C05459=1058.645,309.045,397.535,173.307,35.654,156.681
C05460=1058.639,308.797,397.568,173.303,35.650,156.680
C05461=1058.631,308.551,397.601,173.300,35.645,156.679
C05462=1058.625,308.302,397.633,173.297,35.642,156.679
C05463=1058.618,308.054,397.666,173.293,35.638,156.678
C05464=1058.612,307.806,397.699,173.290,35.634,156.677
C05465=1058.606,307.559,397.731,173.287,35.630,156.676
C05466=1058.600,307.311,397.764,173.283,35.626,156.675
C05467=1058.593,307.064,397.797,173.280,35.622,156.674
C05468=1058.586,306.815,397.830,173.277,35.617,156.673
C05469=1058.579,306.568,397.862,173.274,35.613,156.672
C05470=1058.573,306.320,397.895,173.271,35.609,156.672
C05471=1058.567,306.073,397.928,173.267,35.605,156.671
C05472=1058.560,305.825,397.960,173.264,35.601,156.670
C05473=1058.554,305.578,397.993,173.260,35.598,156.669
C05474=1058.548,305.329,398.025,173.257,35.594,156.668
C05475=1058.541,305.081,398.058,173.255,35.590,156.667
C05476=1058.534,304.834,398.090,173.251,35.585,156.666
C05477=1058.528,304.586,398.123,173.248,35.581,156.666
C05478=1058.522,304.338,398.155,173.244,35.577,156.665
C05479=1058.515,304.090,398.188,173.241,35.573,156.664
C05480=1058.509,303.842,398.220,173.238,35.569,156.663
C05481=1058.503,303.593,398.254,173.234,35.566,156.662
C05482=1058.496,303.345,398.285,173.232,35.561,156.661
C05483=1058.490,303.097,398.318,173.228,35.557,156.660
C05484=1058.484,302.850,398.351,173.225,35.553,156.660
C05485=1058.478,302.602,398.383,173.222,35.549,156.659
C05486=1058.471,302.354,398.416,173.218,35.545,156.658
C05487=1058.464,302.107,398.448,173.216,35.541,156.657
C05488=1058.458,301.859,398.480,173.213,35.538,156.656
C05489=1058.452,301.611,398.513,173.209,35.533,156.655
C05490=1058.446,301.363,398.545,173.206,35.529,156.655
C05491=1058.440,301.115,398.577,173.202,35.525,156.654
C05492=1058.433,300.867,398.609,173.200,35.521,156.653
C05493=1058.427,300.620,398.642,173.197,35.517,156.652
C05494=1058.420,300.372,398.674,173.193,35.514,156.651
C05495=1058.414,300.124,398.706,173.190,35.509,156.650
C05496=1058.408,299.876,398.739,173.187,35.505,156.649
C05497=1058.401,299.628,398.770,173.184,35.501,156.649
C05498=1058.395,299.380,398.802,173.181,35.497,156.648
C05499=1058.389,299.133,398.835,173.177,35.494,156.647
C05500=1058.383,298.884,398.867,173.174,35.490,156.646
C05501=1058.377,298.638,398.899,173.172,35.485,156.645
C05502=1058.371,298.390,398.931,173.168,35.481,156.644
C05503=1058.364,298.142,398.964,173.165,35.477,156.644
C05504=1058.358,297.894,398.996,173.162,35.474,156.643
C05505=1058.352,297.646,399.027,173.159,35.470,156.642
C05506=1058.345,297.398,399.060,173.156,35.466,156.641
C05507=1058.339,297.150,399.092,173.152,35.461,156.640
C05508=1058.334,296.903,399.124,173.150,35.457,156.639
C05509=1058.327,296.655,399.156,173.147,35.454,156.639
C05510=1058.321,296.407,399.188,173.143,35.450,156.638
C05511=1058.314,296.159,399.219,173.140,35.446,156.637
C05512=1058.308,295.911,399.251,173.138,35.442,156.636
C05513=1058.302,295.663,399.283,173.134,35.438,156.635
C05514=1058.295,295.415,399.315,173.131,35.434,156.635
C05515=1058.289,295.168,399.347,173.128,35.430,156.634
C05516=1058.283,294.919,399.379,173.125,35.426,156.633
C05517=1058.276,294.672,399.410,173.122,35.423,156.632
C05518=1058.270,294.424,399.441,173.119,35.419,156.631
C05519=1058.264,294.176,399.473,173.115,35.415,156.630
C05520=1058.257,293.928,399.505,173.113,35.411,156.630
C05521=1058.250,293.680,399.536,173.110,35.407,156.629
C05522=1058.244,293.432,399.568,173.106,35.403,156.628
C05523=1058.238,293.185,399.599,173.104,35.399,156.627
C05524=1058.232,292.937,399.631,173.101,35.396,156.626
C05525=1058.226,292.689,399.663,173.097,35.392,156.626
C05526=1058.219,292.441,399.694,173.095,35.388,156.625
C05527=1058.213,292.193,399.726,173.092,35.384,156.624
C05528=1058.206,291.945,399.758,173.088,35.380,156.623
C05529=1058.200,291.697,399.789,173.086,35.376,156.622
C05530=1058.194,291.457,399.820,173.083,35.373,156.622
C05531=1058.188,291.217,399.850,173.079,35.369,156.621
C05532=1058.182,290.976,399.881,173.077,35.365,156.620
C05533=1058.175,290.736,399.911,173.074,35.362,156.619
C05534=1058.169,290.496,399.942,173.071,35.358,156.619
C05535=1058.163,290.255,399.972,173.068,35.354,156.618
C05536=1058.156,290.015,400.002,173.065,35.350,156.617
C05537=1058.151,289.774,400.033,173.062,35.347,156.616
C05538=1058.144,289.527,400.064,173.059,35.343,156.615
C05539=1058.138,289.279,400.095,173.057,35.339,156.615
C05540=1058.132,289.031,400.128,173.053,35.335,156.614
C05541=1058.126,288.783,400.158,173.050,35.332,156.613
C05542=1058.119,288.535,400.189,173.048,35.327,156.612
C05543=1058.112,288.287,400.221,173.044,35.324,156.611
C05544=1058.106,288.039,400.251,173.041,35.320,156.611
C05545=1058.100,287.791,400.283,173.039,35.316,156.610
C05546=1058.094,287.543,400.315,173.035,35.313,156.609
C05547=1058.088,287.295,400.345,173.032,35.309,156.608
C05548=1058.081,287.047,400.377,173.030,35.305,156.607
C05549=1058.075,286.800,400.408,173.026,35.301,156.607
C05550=1058.068,286.551,400.438,173.024,35.297,156.606
C05551=1058.062,286.303,400.470,173.021,35.294,156.605
C05552=1058.056,286.055,400.500,173.017,35.290,156.604
C05553=1058.049,285.807,400.532,173.015,35.286,156.604
C05554=1058.042,285.560,400.563,173.012,35.282,156.603
C05555=1058.036,285.312,400.593,173.008,35.278,156.602
C05556=1058.030,285.064,400.625,173.006,35.275,156.601
C05557=1058.023,284.815,400.656,173.003,35.271,156.600
C05558=1058.017,284.568,400.687,173.001,35.267,156.600
C05559=1058.011,284.320,400.717,172.997,35.263,156.599
C05560=1058.004,284.071,400.748,172.994,35.260,156.598
C05561=1057.998,283.824,400.779,172.992,35.256,156.597
C05562=1057.992,283.575,400.810,172.988,35.252,156.596
C05563=1057.986,283.328,400.841,172.986,35.248,156.596
C05564=1057.979,283.080,400.872,172.983,35.245,156.595
C05565=1057.973,282.832,400.903,172.980,35.241,156.594
C05566=1057.967,282.584,400.933,172.977,35.237,156.593
C05567=1057.960,282.335,400.964,172.974,35.233,156.593
C05568=1057.954,282.088,400.995,172.971,35.229,156.592
C05569=1057.948,281.840,401.026,172.968,35.226,156.591
C05570=1057.942,281.592,401.056,172.966,35.222,156.590
C05571=1057.935,281.344,401.088,172.962,35.218,156.590
C05572=1057.929,281.096,401.118,172.960,35.215,156.589
C05573=1057.923,280.848,401.149,172.957,35.210,156.588
C05574=1057.917,280.600,401.179,172.955,35.207,156.587
C05575=1057.910,280.352,401.211,172.951,35.203,156.586
C05576=1057.905,280.104,401.241,172.949,35.199,156.586
C05577=1057.898,279.856,401.272,172.946,35.196,156.585
C05578=1057.892,279.608,401.302,172.942,35.192,156.584
C05579=1057.885,279.359,401.332,172.940,35.188,156.583
C05580=1057.879,279.112,401.364,172.937,35.184,156.583
C05581=1057.873,278.864,401.394,172.934,35.181,156.582
C05582=1057.866,278.615,401.425,172.931,35.177,156.581
C05583=1057.860,278.368,401.454,172.929,35.173,156.580
C05584=1057.853,278.119,401.485,172.926,35.170,156.580
C05585=1057.847,277.871,401.515,172.923,35.165,156.579
C05586=1057.842,277.637,401.544,172.920,35.162,156.578
C05587=1057.836,277.401,401.573,172.918,35.159,156.577
C05588=1057.830,277.166,401.602,172.915,35.155,156.577
C05589=1057.824,276.932,401.631,172.912,35.152,156.576
C05590=1057.817,276.697,401.659,172.910,35.148,156.575
C05591=1057.811,276.462,401.688,172.907,35.145,156.574
C05592=1057.806,276.227,401.717,172.904,35.141,156.574
C05593=1057.800,275.992,401.745,172.902,35.138,156.573
C05594=1057.794,275.744,401.776,172.899,35.134,156.572
C05595=1057.787,275.496,401.806,172.896,35.130,156.571
C05596=1057.781,275.248,401.837,172.893,35.126,156.571
C05597=1057.775,275.000,401.867,172.891,35.123,156.570
C05598=1057.764,274.601,401.916,172.886,35.117,156.569
C05599=1057.754,274.203,401.964,172.882,35.111,156.568
C05600=1057.744,273.805,402.012,172.877,35.105,156.566
C05601=1057.734,273.406,402.060,172.873,35.099,156.565
C05602=1057.728,273.158,402.091,172.870,35.095,156.564
C05603=1057.722,272.911,402.121,172.867,35.091,156.564
C05604=1057.715,272.662,402.151,172.865,35.088,156.563
C05605=1057.710,272.414,402.181,172.862,35.084,156.562
C05606=1057.703,272.166,402.211,172.860,35.081,156.561
C05607=1057.697,271.918,402.241,172.856,35.076,156.560
C05608=1057.690,271.670,402.270,172.854,35.073,156.560
C05609=1057.684,271.421,402.301,172.851,35.069,156.559
C05610=1057.678,271.173,402.331,172.849,35.066,156.558
C05611=1057.672,270.926,402.361,172.845,35.062,156.558
C05612=1057.665,270.677,402.391,172.843,35.058,156.557
C05613=1057.659,270.429,402.421,172.841,35.054,156.556
C05614=1057.653,270.181,402.450,172.837,35.051,156.555
C05615=1057.646,269.933,402.481,172.835,35.047,156.555
C05616=1057.640,269.685,402.510,172.832,35.044,156.554
C05617=1057.634,269.437,402.540,172.830,35.040,156.553
C05618=1057.627,269.188,402.570,172.826,35.036,156.552
C05619=1057.621,268.940,402.600,172.824,35.032,156.552
C05620=1057.615,268.692,402.630,172.822,35.029,156.551
C05621=1057.609,268.444,402.659,172.818,35.025,156.550
C05622=1057.602,268.196,402.689,172.816,35.021,156.549
C05623=1057.596,267.948,402.718,172.813,35.018,156.549
C05624=1057.590,267.700,402.749,172.811,35.014,156.548
C05625=1057.583,267.451,402.778,172.808,35.010,156.547
C05626=1057.577,267.204,402.808,172.805,35.007,156.546
C05627=1057.571,266.955,402.838,172.803,35.003,156.546
C05628=1057.565,266.708,402.867,172.800,35.000,156.545
C05629=1057.558,266.459,402.897,172.797,34.995,156.544
C05630=1057.552,266.210,402.926,172.795,34.992,156.543
C05631=1057.546,265.963,402.956,172.792,34.988,156.543
C05632=1057.540,265.715,402.985,172.790,34.985,156.542
C05633=1057.533,265.466,403.016,172.786,34.981,156.541
C05634=1057.527,265.218,403.045,172.784,34.978,156.540
C05635=1057.521,264.970,403.074,172.782,34.973,156.540
C05636=1057.515,264.722,403.104,172.778,34.970,156.539
C05637=1057.509,264.474,403.133,172.776,34.966,156.538
C05638=1057.502,264.225,403.163,172.774,34.963,156.537
C05639=1057.496,263.977,403.192,172.771,34.959,156.537
C05640=1057.490,263.729,403.222,172.768,34.956,156.536
C05641=1057.483,263.481,403.251,172.766,34.951,156.535
C05642=1057.476,263.165,403.288,172.763,34.947,156.534
C05643=1057.468,262.850,403.326,172.760,34.942,156.533
C05644=1057.460,262.534,403.363,172.756,34.938,156.532
C05645=1057.451,262.219,403.400,172.753,34.933,156.532
C05646=1057.444,261.971,403.430,172.750,34.930,156.531
C05647=1057.438,261.722,403.459,172.747,34.926,156.530
C05648=1057.432,261.474,403.488,172.745,34.923,156.529
C05649=1057.425,261.226,403.517,172.742,34.919,156.529
C05650=1057.418,260.977,403.546,172.740,34.915,156.528
C05651=1057.412,260.729,403.575,172.737,34.912,156.527
C05652=1057.406,260.481,403.604,172.734,34.908,156.526
C05653=1057.400,260.233,403.633,172.732,34.905,156.526
C05654=1057.393,259.985,403.662,172.730,34.901,156.525
C05655=1057.387,259.737,403.691,172.726,34.897,156.524
C05656=1057.380,259.488,403.721,172.724,34.893,156.523
C05657=1057.374,259.240,403.750,172.722,34.890,156.523
C05658=1057.368,258.992,403.779,172.719,34.886,156.522
C05659=1057.362,258.743,403.808,172.716,34.883,156.521
C05660=1057.355,258.495,403.837,172.714,34.879,156.521
C05661=1057.349,258.247,403.866,172.711,34.875,156.520
C05662=1057.343,257.999,403.895,172.709,34.872,156.519
C05663=1057.336,257.751,403.923,172.706,34.868,156.518
C05664=1057.329,257.502,403.953,172.703,34.865,156.518
C05665=1057.323,257.254,403.981,172.701,34.861,156.517
C05666=1057.317,257.006,404.010,172.699,34.857,156.516
C05667=1057.311,256.757,404.039,172.695,34.854,156.516
C05668=1057.304,256.509,404.068,172.693,34.850,156.515
C05669=1057.298,256.261,404.097,172.691,34.847,156.514
C05670=1057.292,256.013,404.126,172.689,34.843,156.513
C05671=1057.286,255.765,404.155,172.685,34.839,156.513
C05672=1057.280,255.516,404.184,172.683,34.836,156.512
C05673=1057.273,255.268,404.213,172.681,34.832,156.511
C05674=1057.266,255.020,404.241,172.679,34.828,156.510
C05675=1057.260,254.772,404.270,172.675,34.825,156.510
C05676=1057.254,254.523,404.299,172.673,34.821,156.509
C05677=1057.248,254.275,404.328,172.671,34.817,156.508
C05678=1057.242,254.027,404.357,172.669,34.814,156.508
C05679=1057.235,253.779,404.386,172.666,34.810,156.507
C05680=1057.230,253.530,404.414,172.663,34.807,156.506
C05681=1057.223,253.282,404.443,172.661,34.803,156.505
C05682=1057.217,253.034,404.472,172.659,34.799,156.505
C05683=1057.210,252.785,404.500,172.656,34.796,156.504
C05684=1057.204,252.537,404.529,172.653,34.792,156.503
C05685=1057.198,252.289,404.557,172.651,34.788,156.502
C05686=1057.192,252.040,404.586,172.649,34.784,156.502
C05687=1057.186,251.792,404.615,172.646,34.781,156.501
C05688=1057.180,251.544,404.644,172.643,34.777,156.500
C05689=1057.173,251.295,404.673,172.641,34.774,156.500
C05690=1057.167,251.047,404.700,172.639,34.770,156.499
C05691=1057.161,250.799,404.729,172.637,34.766,156.498
C05692=1057.155,250.551,404.758,172.633,34.762,156.497
C05693=1057.149,250.303,404.786,172.631,34.759,156.497
C05694=1057.143,250.068,404.814,172.629,34.755,156.496
C05695=1057.137,249.835,404.841,172.627,34.752,156.495
C05696=1057.131,249.601,404.868,172.625,34.748,156.494
C05697=1057.125,249.367,404.894,172.622,34.745,156.494
C05698=1057.120,249.133,404.921,172.620,34.741,156.493
C05699=1057.114,248.900,404.948,172.618,34.738,156.492
C05700=1057.108,248.665,404.975,172.616,34.735,156.492
C05701=1057.103,248.431,405.002,172.613,34.731,156.491
C05702=1057.096,248.183,405.030,172.611,34.727,156.490
C05703=1057.090,247.935,405.058,172.608,34.724,156.490
C05704=1057.084,247.686,405.087,172.606,34.720,156.489
C05705=1057.078,247.438,405.116,172.604,34.716,156.488
C05706=1057.072,247.189,405.144,172.601,34.712,156.487
C05707=1057.066,246.941,405.172,172.599,34.709,156.487
C05708=1057.060,246.694,405.201,172.597,34.705,156.486
C05709=1057.054,246.445,405.229,172.594,34.701,156.485
C05710=1057.048,246.196,405.257,172.591,34.697,156.484
C05711=1057.041,245.948,405.286,172.589,34.694,156.484
C05712=1057.035,245.699,405.314,172.587,34.690,156.483
C05713=1057.029,245.451,405.342,172.585,34.687,156.482
C05714=1057.023,245.203,405.370,172.583,34.683,156.481
C05715=1057.017,244.955,405.399,172.579,34.679,156.481
C05716=1057.010,244.706,405.426,172.577,34.676,156.480
C05717=1057.004,244.458,405.455,172.575,34.672,156.479
C05718=1056.998,244.209,405.483,172.573,34.668,156.479
C05719=1056.992,243.961,405.510,172.570,34.664,156.478
C05720=1056.986,243.713,405.539,172.568,34.661,156.477
C05721=1056.979,243.465,405.567,172.566,34.657,156.476
C05722=1056.973,243.216,405.596,172.563,34.654,156.476
C05723=1056.967,242.967,405.623,172.561,34.650,156.475
C05724=1056.961,242.719,405.651,172.558,34.646,156.474
C05725=1056.955,242.471,405.679,172.556,34.643,156.474
C05726=1056.949,242.222,405.707,172.554,34.639,156.473
C05727=1056.942,241.974,405.736,172.552,34.635,156.472
C05728=1056.936,241.726,405.764,172.549,34.631,156.471
C05729=1056.930,241.478,405.791,172.547,34.628,156.471
C05730=1056.924,241.229,405.820,172.544,34.624,156.470
C05731=1056.917,240.981,405.847,172.542,34.620,156.469
C05732=1056.911,240.733,405.875,172.540,34.617,156.468
C05733=1056.905,240.484,405.903,172.537,34.613,156.468
C05734=1056.898,240.236,405.931,172.535,34.610,156.467
C05735=1056.892,239.987,405.959,172.533,34.606,156.466
C05736=1056.886,239.739,405.987,172.531,34.602,156.466
C05737=1056.880,239.490,406.014,172.529,34.599,156.465
C05738=1056.873,239.242,406.041,172.526,34.595,156.464
C05739=1056.867,238.993,406.070,172.523,34.592,156.463
C05740=1056.861,238.745,406.097,172.521,34.588,156.463
C05741=1056.854,238.497,406.125,172.519,34.584,156.462
C05742=1056.849,238.248,406.153,172.516,34.580,156.461
C05743=1056.842,238.000,406.181,172.514,34.577,156.460
C05744=1056.836,237.752,406.208,172.512,34.573,156.460
C05745=1056.829,237.503,406.236,172.510,34.569,156.459
C05746=1056.823,237.254,406.264,172.508,34.566,156.458
C05747=1056.817,237.006,406.291,172.505,34.562,156.458
C05748=1056.811,236.758,406.319,172.503,34.558,156.457
C05749=1056.804,236.509,406.346,172.501,34.555,156.456
C05750=1056.799,236.273,406.372,172.499,34.551,156.455
C05751=1056.792,236.036,406.399,172.497,34.548,156.455
C05752=1056.787,235.799,406.426,172.494,34.544,156.454
C05753=1056.781,235.562,406.452,172.492,34.541,156.453
C05754=1056.775,235.325,406.478,172.490,34.537,156.453
C05755=1056.769,235.088,406.505,172.488,34.534,156.452
C05756=1056.763,234.850,406.530,172.486,34.530,156.451
C05757=1056.758,234.614,406.556,172.484,34.527,156.451
C05758=1056.751,234.365,406.584,172.481,34.523,156.450
C05759=1056.744,234.117,406.612,172.479,34.519,156.449
C05760=1056.739,233.868,406.639,172.477,34.516,156.448
C05761=1056.732,233.620,406.667,172.475,34.512,156.448
C05762=1056.726,233.372,406.694,172.473,34.508,156.447
C05763=1056.720,233.123,406.721,172.470,34.504,156.446
C05764=1056.714,232.875,406.748,172.468,34.501,156.446
C05765=1056.708,232.627,406.777,172.466,34.497,156.445
C05766=1056.702,232.377,406.804,172.464,34.493,156.444
C05767=1056.696,232.130,406.831,172.462,34.490,156.443
C05768=1056.689,231.881,406.858,172.459,34.486,156.443
C05769=1056.683,231.633,406.885,172.457,34.483,156.442
C05770=1056.677,231.384,406.912,172.455,34.479,156.441
C05771=1056.670,231.135,406.940,172.453,34.475,156.440
C05772=1056.664,230.887,406.967,172.451,34.471,156.440
C05773=1056.658,230.639,406.995,172.448,34.467,156.439
C05774=1056.652,230.390,407.021,172.446,34.464,156.438
C05775=1056.645,230.142,407.049,172.444,34.460,156.438
C05776=1056.639,229.893,407.076,172.442,34.457,156.437
C05777=1056.633,229.645,407.104,172.440,34.453,156.436
C05778=1056.628,229.396,407.131,172.437,34.449,156.435
C05779=1056.621,229.148,407.158,172.435,34.445,156.435
C05780=1056.614,228.900,407.184,172.433,34.441,156.434
C05781=1056.608,228.651,407.212,172.431,34.438,156.433
C05782=1056.601,228.402,407.239,172.429,34.434,156.433
C05783=1056.596,228.154,407.266,172.426,34.431,156.432
C05784=1056.589,227.906,407.294,172.424,34.427,156.431
C05785=1056.583,227.657,407.320,172.422,34.423,156.430
C05786=1056.577,227.408,407.347,172.420,34.420,156.430
C05787=1056.570,227.161,407.374,172.418,34.416,156.429
C05788=1056.564,226.912,407.401,172.415,34.412,156.428
C05789=1056.558,226.663,407.428,172.413,34.408,156.427
C05790=1056.551,226.415,407.455,172.411,34.405,156.427
C05791=1056.545,226.167,407.482,172.409,34.401,156.426
C05792=1056.539,225.917,407.509,172.407,34.397,156.425
C05793=1056.533,225.669,407.536,172.405,34.394,156.425
C05794=1056.526,225.421,407.563,172.402,34.390,156.424
C05795=1056.520,225.173,407.589,172.400,34.386,156.423
C05796=1056.514,224.924,407.616,172.398,34.383,156.422
C05797=1056.508,224.675,407.643,172.396,34.379,156.422
C05798=1056.502,224.427,407.670,172.394,34.375,156.421
C05799=1056.495,224.178,407.697,172.391,34.371,156.420
C05800=1056.489,223.930,407.724,172.389,34.368,156.420
C05801=1056.482,223.681,407.751,172.387,34.364,156.419
C05802=1056.477,223.433,407.777,172.385,34.360,156.418
C05803=1056.471,223.185,407.804,172.383,34.356,156.417
C05804=1056.465,222.935,407.831,172.382,34.353,156.417
C05805=1056.459,222.687,407.857,172.379,34.349,156.416
C05806=1056.452,222.446,407.884,172.377,34.345,156.415
C05807=1056.447,222.206,407.910,172.375,34.342,156.414
C05808=1056.440,221.964,407.936,172.373,34.338,156.414
C05809=1056.434,221.724,407.962,172.371,34.335,156.413
C05810=1056.428,221.483,407.988,172.368,34.331,156.412
C05811=1056.423,221.242,408.013,172.366,34.327,156.412
C05812=1056.416,221.001,408.039,172.365,34.324,156.411
C05813=1056.411,220.760,408.065,172.363,34.320,156.410
C05814=1056.404,220.512,408.091,172.361,34.316,156.410
C05815=1056.398,220.263,408.118,172.359,34.313,156.409
C05816=1056.391,220.015,408.144,172.356,34.309,156.408
C05817=1056.385,219.766,408.171,172.354,34.305,156.407
C05818=1056.379,219.518,408.197,172.352,34.301,156.407
C05819=1056.372,219.269,408.224,172.350,34.298,156.406
C05820=1056.366,219.021,408.250,172.348,34.294,156.405
C05821=1056.360,218.773,408.276,172.347,34.290,156.404
C05822=1056.353,218.524,408.304,172.344,34.287,156.404
C05823=1056.347,218.276,408.330,172.342,34.283,156.403
C05824=1056.341,218.027,408.356,172.340,34.279,156.402
C05825=1056.335,217.778,408.383,172.338,34.275,156.402
C05826=1056.329,217.530,408.409,172.336,34.272,156.401
C05827=1056.323,217.281,408.435,172.334,34.268,156.400
C05828=1056.316,217.032,408.462,172.331,34.264,156.399
C05829=1056.310,216.784,408.488,172.329,34.260,156.399
C05830=1056.303,216.536,408.514,172.328,34.257,156.398
C05831=1056.297,216.287,408.541,172.326,34.253,156.397
C05832=1056.291,216.038,408.567,172.324,34.249,156.396
C05833=1056.285,215.790,408.593,172.321,34.246,156.396
C05834=1056.279,215.542,408.619,172.319,34.241,156.395
C05835=1056.272,215.293,408.646,172.317,34.238,156.394
C05836=1056.266,215.044,408.672,172.315,34.234,156.394
C05837=1056.260,214.796,408.698,172.314,34.230,156.393
C05838=1056.254,214.548,408.724,172.312,34.226,156.392
C05839=1056.247,214.299,408.751,172.309,34.223,156.391
C05840=1056.241,214.050,408.777,172.307,34.219,156.391
C05841=1056.235,213.802,408.803,172.305,34.215,156.390
C05842=1056.229,213.554,408.829,172.303,34.211,156.389
C05843=1056.223,213.304,408.856,172.302,34.207,156.388
C05844=1056.217,213.056,408.882,172.300,34.204,156.388
C05845=1056.210,212.808,408.908,172.297,34.200,156.387
C05846=1056.204,212.559,408.934,172.295,34.196,156.386
C05847=1056.198,212.311,408.960,172.293,34.192,156.385
C05848=1056.191,212.062,408.987,172.291,34.189,156.385
C05849=1056.186,211.813,409.013,172.290,34.184,156.384
C05850=1056.179,211.565,409.039,172.288,34.181,156.383
C05851=1056.173,211.316,409.064,172.286,34.177,156.383
C05852=1056.167,211.067,409.091,172.283,34.174,156.382
C05853=1056.160,210.819,409.117,172.281,34.169,156.381
C05854=1056.154,210.570,409.143,172.279,34.166,156.380
C05855=1056.148,210.322,409.169,172.278,34.162,156.380
C05856=1056.142,210.073,409.195,172.276,34.158,156.379
C05857=1056.135,209.824,409.221,172.274,34.154,156.378
C05858=1056.129,209.576,409.247,172.271,34.150,156.377
C05859=1056.123,209.327,409.273,172.269,34.147,156.377
C05860=1056.117,209.079,409.298,172.268,34.143,156.376
C05861=1056.110,208.831,409.324,172.266,34.139,156.375
C05862=1056.104,208.592,409.350,172.264,34.135,156.374
C05863=1056.099,208.354,409.375,172.262,34.132,156.374
C05864=1056.092,208.116,409.399,172.260,34.128,156.373
C05865=1056.087,207.877,409.424,172.258,34.124,156.372
C05866=1056.081,207.639,409.448,172.256,34.121,156.372
C05867=1056.075,207.400,409.473,172.255,34.117,156.371
C05868=1056.069,207.162,409.498,172.253,34.114,156.370
C05869=1056.062,206.924,409.522,172.251,34.110,156.370
C05870=1056.037,205.873,409.627,172.050,34.020,156.356
C05871=1056.031,205.624,409.652,172.048,34.017,156.356
C05872=1056.025,205.376,409.677,172.045,34.014,156.355
C05873=1056.020,205.127,409.702,172.043,34.011,156.355
C05874=1056.013,204.878,409.727,172.041,34.008,156.354
C05875=1056.008,204.630,409.752,172.038,34.005,156.354
C05876=1056.001,204.381,409.776,172.036,34.002,156.353
C05877=1055.996,204.133,409.801,172.034,33.999,156.353
C05878=1055.990,203.884,409.826,172.031,33.996,156.352
C05879=1055.984,203.635,409.851,172.028,33.993,156.352
C05880=1055.978,203.387,409.876,172.026,33.990,156.351
C05881=1055.972,203.138,409.900,172.024,33.987,156.351
C05882=1055.966,202.888,409.925,172.021,33.984,156.350
C05883=1055.961,202.640,409.950,172.019,33.982,156.350
C05884=1055.954,202.391,409.974,172.017,33.978,156.349
C05885=1055.948,202.143,409.999,172.015,33.975,156.348
C05886=1055.943,201.894,410.023,172.012,33.972,156.348
C05887=1055.937,201.645,410.048,172.010,33.970,156.347
C05888=1055.930,201.397,410.072,172.008,33.967,156.347
C05889=1055.924,201.148,410.097,172.005,33.964,156.346
C05890=1055.918,200.899,410.122,172.002,33.961,156.346
C05891=1055.912,200.651,410.146,172.000,33.958,156.345
C05892=1055.906,200.402,410.171,171.998,33.955,156.345
C05893=1055.900,200.153,410.194,171.995,33.953,156.344
C05894=1055.894,199.904,410.219,171.993,33.950,156.344
C05895=1055.888,199.655,410.244,171.991,33.947,156.343
C05896=1055.882,199.407,410.268,171.989,33.944,156.343
C05897=1055.876,199.158,410.293,171.986,33.941,156.342
C05898=1055.870,198.910,410.316,171.984,33.938,156.342
C05899=1055.864,198.661,410.342,171.982,33.936,156.341
C05900=1055.857,198.412,410.366,171.980,33.933,156.341
C05901=1055.852,198.163,410.390,171.976,33.930,156.340
C05902=1055.845,197.914,410.414,171.974,33.927,156.340
C05903=1055.840,197.666,410.438,171.972,33.924,156.339
C05904=1055.834,197.416,410.463,171.970,33.921,156.339
C05905=1055.828,197.169,410.487,171.967,33.919,156.338
C05906=1055.822,196.919,410.512,171.965,33.916,156.338
C05907=1055.815,196.671,410.536,171.963,33.913,156.337
C05908=1055.810,196.422,410.560,171.961,33.910,156.337
C05909=1055.803,196.173,410.584,171.958,33.907,156.336
C05910=1055.798,195.924,410.608,171.956,33.904,156.336
C05911=1055.791,195.675,410.632,171.954,33.902,156.335
C05912=1055.786,195.427,410.657,171.952,33.899,156.335
C05913=1055.779,195.178,410.681,171.949,33.896,156.334
C05914=1055.774,194.929,410.705,171.946,33.893,156.334
C05915=1055.768,194.680,410.729,171.944,33.891,156.333
C05916=1055.762,194.432,410.753,171.942,33.887,156.333
C05917=1055.756,194.183,410.777,171.940,33.885,156.332
C05918=1055.750,193.934,410.801,171.937,33.882,156.332
C05919=1055.744,193.686,410.825,171.935,33.879,156.331
C05920=1055.738,193.437,410.850,171.933,33.876,156.331
C05921=1055.732,193.188,410.873,171.931,33.874,156.330
C05922=1055.726,192.939,410.898,171.929,33.870,156.330
C05923=1055.720,192.691,410.922,171.926,33.868,156.329
C05924=1055.714,192.441,410.946,171.924,33.865,156.329
C05925=1055.708,192.193,410.970,171.922,33.862,156.328
C05926=1055.703,191.945,410.994,171.920,33.860,156.328
C05927=1055.696,191.696,411.018,171.917,33.857,156.327
C05928=1055.691,191.447,411.042,171.915,33.854,156.327
C05929=1055.685,191.198,411.067,171.912,33.851,156.326
C05930=1055.679,190.949,411.091,171.910,33.848,156.326
C05931=1055.673,190.665,411.118,171.908,33.845,156.325
C05932=1055.666,190.381,411.145,171.905,33.842,156.325
C05933=1055.659,190.097,411.173,171.903,33.839,156.324
C05934=1055.653,189.813,411.200,171.900,33.836,156.323
C05935=1055.647,189.564,411.223,171.898,33.833,156.323
C05936=1055.641,189.316,411.248,171.896,33.830,156.322
C05937=1055.635,189.067,411.272,171.894,33.827,156.322
C05938=1055.630,188.818,411.295,171.892,33.824,156.321
C05939=1055.624,188.569,411.319,171.890,33.822,156.321
C05940=1055.618,188.320,411.344,171.887,33.819,156.320
C05941=1055.612,188.072,411.367,171.884,33.816,156.320
C05942=1055.606,187.824,411.391,171.882,33.813,156.319
C05943=1055.600,187.574,411.415,171.880,33.811,156.319
C05944=1055.594,187.325,411.438,171.878,33.807,156.318
C05945=1055.589,187.077,411.463,171.876,33.805,156.318
C05946=1055.583,186.828,411.486,171.874,33.802,156.317
C05947=1055.577,186.579,411.510,171.871,33.799,156.317
C05948=1055.571,186.330,411.534,171.869,33.797,156.316
C05949=1055.566,186.081,411.558,171.867,33.794,156.316
C05950=1055.559,185.832,411.582,171.865,33.791,156.315
C05951=1055.553,185.584,411.605,171.863,33.788,156.315
C05952=1055.548,185.335,411.629,171.861,33.785,156.314
C05953=1055.542,185.086,411.652,171.859,33.783,156.314
C05954=1055.537,184.838,411.677,171.857,33.780,156.313
C05955=1055.531,184.588,411.700,171.854,33.777,156.313
C05956=1055.525,184.340,411.724,171.851,33.774,156.312
C05957=1055.520,184.091,411.747,171.849,33.771,156.312
C05958=1055.513,183.842,411.771,171.847,33.769,156.311
C05959=1055.507,183.593,411.794,171.845,33.766,156.311
C05960=1055.500,183.345,411.817,171.843,33.764,156.311
C05961=1055.494,183.095,411.841,171.841,33.761,156.310
C05962=1055.488,182.847,411.864,171.839,33.759,156.310
C05963=1055.482,182.598,411.887,171.837,33.756,156.309
C05964=1055.476,182.349,411.911,171.834,33.754,156.309
C05965=1055.470,182.100,411.934,171.832,33.751,156.308
C05966=1055.464,181.851,411.957,171.830,33.748,156.308
C05967=1055.458,181.602,411.981,171.828,33.745,156.307
C05968=1055.452,181.353,412.004,171.826,33.743,156.307
C05969=1055.446,181.105,412.028,171.824,33.740,156.306
C05970=1055.440,180.856,412.051,171.822,33.738,156.306
C05971=1055.434,180.607,412.074,171.820,33.735,156.306
C05972=1055.428,180.358,412.098,171.817,33.733,156.305
C05973=1055.421,180.110,412.120,171.814,33.730,156.305
C05974=1055.415,179.860,412.143,171.812,33.727,156.304
C05975=1055.409,179.612,412.167,171.810,33.725,156.304
C05976=1055.403,179.363,412.190,171.808,33.722,156.303
C05977=1055.397,179.114,412.213,171.806,33.719,156.303
C05978=1055.391,178.865,412.237,171.804,33.717,156.302
C05979=1055.385,178.616,412.260,171.802,33.714,156.302
C05980=1055.379,178.367,412.283,171.800,33.712,156.301
C05981=1055.374,178.119,412.306,171.798,33.709,156.301
C05982=1055.366,177.870,412.329,171.796,33.707,156.301
C05983=1055.361,177.621,412.352,171.793,33.704,156.300
C05984=1055.355,177.372,412.375,171.791,33.702,156.300
C05985=1055.349,177.123,412.398,171.789,33.698,156.299
C05986=1055.343,176.875,412.422,171.787,33.696,156.299
C05987=1055.337,176.625,412.445,171.785,33.693,156.298
C05988=1055.331,176.376,412.468,171.783,33.691,156.298
C05989=1055.325,176.127,412.491,171.781,33.688,156.297
C05990=1055.319,175.879,412.513,171.779,33.686,156.297
C05991=1055.313,175.631,412.537,171.777,33.683,156.296
C05992=1055.307,175.382,412.560,171.774,33.681,156.296
C05993=1055.301,175.132,412.583,171.772,33.678,156.296
C05994=1055.295,174.883,412.606,171.770,33.676,156.295
C05995=1055.288,174.599,412.632,171.767,33.672,156.295
C05996=1055.282,174.315,412.659,171.765,33.669,156.294
C05997=1055.275,174.030,412.684,171.763,33.667,156.294
C05998=1055.268,173.746,412.711,171.760,33.664,156.293
C05999=1055.262,173.497,412.734,171.758,33.661,156.293
C06000=1055.256,173.249,412.757,171.756,33.658,156.292
C06001=1055.250,173.000,412.780,171.754,33.656,156.292
C06002=1055.244,172.750,412.803,171.752,33.653,156.291
C06003=1055.238,172.501,412.826,171.750,33.651,156.291
C06004=1055.232,172.253,412.848,171.748,33.648,156.290
C06005=1055.226,172.004,412.871,171.746,33.645,156.290
C06006=1055.220,171.755,412.894,171.744,33.643,156.289
C06007=1055.215,171.506,412.917,171.742,33.640,156.289
C06008=1055.209,171.257,412.940,171.740,33.638,156.288
C06009=1055.202,171.008,412.962,171.738,33.635,156.288
C06010=1055.197,170.760,412.985,171.736,33.632,156.288
C06011=1055.191,170.511,413.008,171.734,33.630,156.287
C06012=1055.185,170.262,413.031,171.732,33.627,156.287
C06013=1055.179,170.013,413.054,171.729,33.625,156.286
C06014=1055.174,169.764,413.077,171.727,33.622,156.286
C06015=1055.167,169.515,413.099,171.725,33.620,156.285
C06016=1055.162,169.266,413.122,171.723,33.617,156.285
C06017=1055.156,169.018,413.145,171.721,33.615,156.284
C06018=1055.150,168.769,413.168,171.719,33.611,156.284
C06019=1055.145,168.519,413.191,171.717,33.609,156.283
C06020=1055.138,168.271,413.213,171.715,33.606,156.283
C06021=1055.132,168.022,413.236,171.713,33.604,156.283
C06022=1055.127,167.773,413.259,171.711,33.601,156.282
C06023=1055.121,167.524,413.282,171.709,33.599,156.282
C06024=1055.115,167.275,413.304,171.707,33.596,156.281
C06025=1055.109,167.026,413.327,171.705,33.594,156.281
C06026=1055.103,166.777,413.349,171.703,33.591,156.280
C06027=1055.098,166.528,413.372,171.701,33.589,156.280
C06028=1055.092,166.279,413.395,171.699,33.586,156.280
C06029=1055.085,166.030,413.417,171.697,33.583,156.279
C06030=1055.080,165.782,413.440,171.695,33.581,156.279
C06031=1055.074,165.532,413.463,171.693,33.578,156.278
C06032=1055.069,165.283,413.486,171.692,33.575,156.278
C06033=1055.063,165.035,413.508,171.690,33.573,156.277
C06034=1055.057,164.786,413.531,171.688,33.570,156.277
C06035=1055.052,164.537,413.553,171.686,33.568,156.276
C06036=1055.046,164.288,413.576,171.683,33.565,156.276
C06037=1055.039,164.039,413.598,171.681,33.563,156.275
C06038=1055.034,163.790,413.621,171.679,33.560,156.275
C06039=1055.028,163.541,413.643,171.677,33.557,156.275
C06040=1055.022,163.292,413.666,171.675,33.555,156.274
C06041=1055.016,163.043,413.689,171.673,33.552,156.274
C06042=1055.011,162.795,413.710,171.671,33.550,156.273
C06043=1055.005,162.546,413.733,171.669,33.547,156.273
C06044=1054.999,162.297,413.756,171.667,33.545,156.272
C06045=1054.994,162.048,413.778,171.665,33.542,156.272
C06046=1054.988,161.799,413.801,171.663,33.539,156.271
C06047=1054.982,161.550,413.824,171.661,33.536,156.271
C06048=1054.976,161.301,413.845,171.659,33.534,156.270
C06049=1054.971,161.052,413.868,171.658,33.531,156.270
C06050=1054.965,160.803,413.890,171.656,33.529,156.270
C06051=1054.959,160.554,413.913,171.654,33.526,156.269
C06052=1054.953,160.305,413.935,171.652,33.524,156.269
C06053=1054.947,160.056,413.957,171.650,33.521,156.268
C06054=1054.941,159.807,413.979,171.648,33.519,156.268
C06055=1054.935,159.558,414.002,171.646,33.517,156.267
C06056=1054.929,159.309,414.023,171.644,33.514,156.267
C06057=1054.922,159.060,414.046,171.642,33.512,156.267
C06058=1054.918,158.812,414.068,171.640,33.509,156.266
C06059=1054.911,158.554,414.091,171.638,33.506,156.266
C06060=1054.905,158.297,414.114,171.636,33.504,156.265
C06061=1054.899,158.038,414.137,171.634,33.501,156.265
C06062=1054.892,157.781,414.159,171.632,33.499,156.264
C06063=1054.887,157.532,414.181,171.630,33.496,156.264
C06064=1054.880,157.283,414.204,171.627,33.494,156.263
C06065=1054.874,157.034,414.225,171.625,33.491,156.263
C06066=1054.869,156.785,414.247,171.623,33.489,156.263
C06067=1054.863,156.537,414.270,171.622,33.487,156.262
C06068=1054.857,156.288,414.291,171.620,33.484,156.262
C06069=1054.851,156.039,414.314,171.618,33.482,156.261
C06070=1054.845,155.789,414.336,171.616,33.479,156.261
C06071=1054.839,155.540,414.358,171.614,33.476,156.261
C06072=1054.834,155.292,414.380,171.612,33.474,156.260
C06073=1054.827,155.043,414.402,171.610,33.471,156.260
C06074=1054.821,154.794,414.423,171.608,33.469,156.259
C06075=1054.815,154.545,414.446,171.606,33.467,156.259
C06076=1054.809,154.296,414.468,171.604,33.464,156.258
C06077=1054.804,154.047,414.489,171.602,33.462,156.258
C06078=1054.798,153.798,414.511,171.601,33.459,156.258
C06079=1054.791,153.549,414.533,171.599,33.457,156.257
C06080=1054.786,153.300,414.555,171.597,33.455,156.257
C06081=1054.780,153.051,414.577,171.595,33.452,156.256
C06082=1054.774,152.802,414.598,171.593,33.449,156.256
C06083=1054.767,152.525,414.623,171.591,33.447,156.255
C06084=1054.761,152.249,414.647,171.589,33.444,156.255
C06085=1054.754,151.973,414.671,171.587,33.441,156.254
C06086=1054.748,151.697,414.695,171.585,33.439,156.254
C06087=1054.741,151.448,414.718,171.583,33.436,156.254
C06088=1054.735,151.199,414.739,171.581,33.434,156.253
C06089=1054.730,150.950,414.761,171.579,33.432,156.253
C06090=1054.724,150.701,414.783,171.577,33.429,156.252
C06091=1054.718,150.452,414.804,171.575,33.426,156.252
C06092=1054.712,150.203,414.826,171.573,33.424,156.252
C06093=1054.706,149.955,414.848,171.571,33.421,156.251
C06094=1054.700,149.706,414.870,171.570,33.419,156.251
C06095=1054.693,149.456,414.891,171.568,33.417,156.250
C06096=1054.689,149.208,414.913,171.566,33.414,156.250
C06097=1054.682,148.958,414.935,171.564,33.412,156.249
C06098=1054.676,148.709,414.956,171.562,33.409,156.249
C06099=1054.670,148.460,414.978,171.560,33.407,156.249
C06100=1054.664,148.211,414.999,171.558,33.405,156.248
C06101=1054.658,147.962,415.021,171.556,33.402,156.248
C06102=1054.652,147.713,415.043,171.554,33.400,156.247
C06103=1054.647,147.464,415.064,171.552,33.397,156.247
C06104=1054.640,147.215,415.085,171.550,33.395,156.247
C06105=1054.634,146.966,415.107,171.548,33.392,156.246
C06106=1054.628,146.717,415.129,171.546,33.390,156.246
C06107=1054.623,146.468,415.150,171.544,33.388,156.245
C06108=1054.616,146.219,415.172,171.542,33.385,156.245
C06109=1054.610,145.970,415.193,171.541,33.383,156.245
C06110=1054.605,145.721,415.215,171.539,33.380,156.244
C06111=1054.599,145.472,415.236,171.537,33.378,156.244
C06112=1054.592,145.223,415.258,171.535,33.376,156.243
C06113=1054.587,144.975,415.279,171.533,33.373,156.243
C06114=1054.581,144.725,415.301,171.531,33.371,156.242
C06115=1054.574,144.476,415.322,171.530,33.369,156.242
C06116=1054.569,144.227,415.343,171.528,33.366,156.242
C06117=1054.562,143.978,415.364,171.526,33.364,156.241
C06118=1054.556,143.729,415.386,171.524,33.362,156.241
C06119=1054.551,143.480,415.407,171.522,33.359,156.240
C06120=1054.544,143.231,415.429,171.520,33.356,156.240
C06121=1054.538,142.982,415.450,171.518,33.354,156.240
C06122=1054.533,142.733,415.471,171.517,33.352,156.239
C06123=1054.526,142.448,415.496,171.515,33.349,156.239
C06124=1054.519,142.163,415.520,171.512,33.346,156.238
C06125=1054.513,141.878,415.545,171.510,33.344,156.238
C06126=1054.506,141.593,415.569,171.508,33.340,156.237
C06127=1054.499,141.343,415.590,171.506,33.338,156.237
C06128=1054.494,141.095,415.612,171.505,33.336,156.237
C06129=1054.488,140.846,415.633,171.503,33.333,156.236
C06130=1054.482,140.597,415.654,171.501,33.331,156.236
C06131=1054.476,140.347,415.675,171.499,33.329,156.235
C06132=1054.469,140.098,415.696,171.497,33.326,156.235
C06133=1054.464,139.850,415.718,171.496,33.324,156.234
C06134=1054.458,139.600,415.739,171.494,33.322,156.234
C06135=1054.452,139.352,415.760,171.492,33.319,156.234
C06136=1054.446,139.102,415.782,171.490,33.317,156.233
C06137=1054.440,138.853,415.802,171.488,33.315,156.233
C06138=1054.434,138.604,415.823,171.486,33.312,156.233
C06139=1054.428,138.355,415.845,171.485,33.310,156.232
C06140=1054.423,138.106,415.865,171.483,33.308,156.232
C06141=1054.416,137.857,415.886,171.481,33.305,156.231
C06142=1054.410,137.609,415.908,171.479,33.302,156.231
C06143=1054.404,137.359,415.929,171.477,33.300,156.230
C06144=1054.399,137.110,415.950,171.476,33.298,156.230
C06145=1054.392,136.861,415.970,171.474,33.295,156.230
C06146=1054.386,136.612,415.992,171.472,33.293,156.229
C06147=1054.380,136.363,416.013,171.470,33.291,156.229
C06148=1054.374,136.114,416.033,171.468,33.288,156.229
C06149=1054.368,135.865,416.055,171.467,33.286,156.228
C06150=1054.362,135.615,416.076,171.465,33.284,156.228
C06151=1054.356,135.367,416.096,171.463,33.281,156.227
C06152=1054.350,135.117,416.117,171.461,33.279,156.227
C06153=1054.345,134.869,416.138,171.459,33.277,156.227
C06154=1054.338,134.620,416.159,171.458,33.274,156.226
C06155=1054.332,134.371,416.180,171.456,33.272,156.226
C06156=1054.326,134.121,416.202,171.454,33.270,156.225
C06157=1054.320,133.873,416.222,171.452,33.267,156.225
C06158=1054.314,133.623,416.243,171.450,33.265,156.225
C06159=1054.309,133.374,416.264,171.449,33.263,156.224
C06160=1054.302,133.125,416.285,171.447,33.260,156.224
C06161=1054.297,132.876,416.305,171.445,33.258,156.223
C06162=1054.290,132.627,416.326,171.443,33.255,156.223
C06163=1054.285,132.378,416.347,171.441,33.253,156.223
C06164=1054.279,132.128,416.368,171.439,33.251,156.222
C06165=1054.272,131.880,416.389,171.437,33.248,156.222
C06166=1054.267,131.630,416.409,171.435,33.246,156.221
C06167=1054.260,131.382,416.430,171.433,33.244,156.221
C06168=1054.254,131.132,416.451,171.432,33.241,156.221
C06169=1054.248,130.884,416.471,171.430,33.239,156.220
C06170=1054.242,130.634,416.493,171.428,33.237,156.220
C06171=1054.236,130.386,416.513,171.426,33.235,156.220
C06172=1054.230,130.136,416.533,171.425,33.232,156.219
C06173=1054.224,129.888,416.554,171.423,33.230,156.219
C06174=1054.218,129.638,416.575,171.421,33.228,156.218
C06175=1054.212,129.389,416.595,171.419,33.225,156.218
C06176=1054.205,129.140,416.616,171.417,33.223,156.218
C06177=1054.199,128.891,416.636,171.416,33.221,156.217
C06178=1054.193,128.642,416.656,171.414,33.219,156.217
C06179=1054.188,128.393,416.677,171.412,33.216,156.216
C06180=1054.181,128.144,416.698,171.410,33.214,156.216
C06181=1054.175,127.895,416.719,171.409,33.212,156.216
C06182=1054.169,127.646,416.739,171.407,33.210,156.215
C06183=1054.162,127.397,416.760,171.405,33.207,156.215
C06184=1054.157,127.148,416.780,171.403,33.204,156.214
C06185=1054.151,126.898,416.800,171.401,33.202,156.214
C06186=1054.145,126.649,416.820,171.400,33.200,156.214
C06187=1054.138,126.364,416.844,171.398,33.197,156.213
C06188=1054.131,126.079,416.868,171.396,33.195,156.213
C06189=1054.124,125.793,416.891,171.394,33.192,156.212
C06190=1054.117,125.509,416.915,171.392,33.190,156.212
C06191=1054.111,125.259,416.935,171.390,33.188,156.212
C06192=1054.105,125.010,416.955,171.388,33.185,156.211
C06193=1054.099,124.760,416.976,171.386,33.182,156.211
C06194=1054.093,124.512,416.996,171.385,33.181,156.210
C06195=1054.087,124.263,417.016,171.383,33.178,156.210
C06196=1054.081,124.014,417.037,171.381,33.176,156.210
C06197=1054.075,123.765,417.057,171.379,33.173,156.209
C06198=1054.069,123.516,417.077,171.378,33.171,156.209
C06199=1054.063,123.266,417.098,171.376,33.169,156.208
C06200=1054.057,123.017,417.118,171.374,33.166,156.208
C06201=1054.050,122.768,417.139,171.372,33.164,156.208
C06202=1054.045,122.519,417.159,171.371,33.162,156.207
C06203=1054.039,122.270,417.179,171.369,33.160,156.207
C06204=1054.032,122.020,417.199,171.367,33.157,156.207
C06205=1054.027,121.771,417.220,171.365,33.155,156.206
C06206=1054.021,121.522,417.240,171.364,33.153,156.206
C06207=1054.014,121.274,417.261,171.362,33.150,156.205
C06208=1054.008,121.025,417.281,171.360,33.148,156.205
C06209=1054.003,120.776,417.301,171.359,33.146,156.205
C06210=1053.997,120.527,417.321,171.357,33.144,156.204
C06211=1053.990,120.277,417.342,171.355,33.141,156.204
C06212=1053.985,120.028,417.362,171.353,33.138,156.203
C06213=1053.979,119.779,417.382,171.352,33.137,156.203
C06214=1053.972,119.530,417.403,171.350,33.134,156.203
C06215=1053.966,119.281,417.423,171.348,33.132,156.202
C06216=1053.961,119.032,417.443,171.346,33.129,156.202
C06217=1053.956,118.782,417.462,171.345,33.127,156.201
C06218=1053.949,118.533,417.483,171.343,33.125,156.201
C06219=1053.943,118.284,417.503,171.341,33.122,156.201
C06220=1053.938,118.035,417.523,171.340,33.120,156.200
C06221=1053.932,117.786,417.543,171.338,33.118,156.200
C06222=1053.925,117.537,417.563,171.336,33.115,156.200
C06223=1053.920,117.288,417.584,171.334,33.113,156.199
C06224=1053.914,117.039,417.604,171.333,33.111,156.199
C06225=1053.908,116.790,417.624,171.331,33.108,156.198
C06226=1053.901,116.540,417.644,171.329,33.106,156.198
C06227=1053.896,116.291,417.665,171.328,33.104,156.198
C06228=1053.890,116.042,417.685,171.326,33.101,156.197
C06229=1053.884,115.793,417.704,171.324,33.099,156.197
C06230=1053.878,115.544,417.724,171.323,33.097,156.196
C06231=1053.872,115.294,417.745,171.321,33.095,156.196
C06232=1053.867,115.046,417.765,171.319,33.092,156.196
C06233=1053.861,114.797,417.785,171.317,33.089,156.195
C06234=1053.855,114.548,417.805,171.316,33.087,156.195
C06235=1053.849,114.299,417.824,171.314,33.085,156.194
C06236=1053.843,114.049,417.845,171.312,33.082,156.194
C06237=1053.837,113.800,417.865,171.311,33.080,156.194
C06238=1053.831,113.551,417.885,171.309,33.078,156.193
C06239=1053.825,113.302,417.904,171.307,33.076,156.193
C06240=1053.819,113.052,417.924,171.306,33.073,156.193
C06241=1053.813,112.803,417.944,171.304,33.071,156.192
C06242=1053.807,112.554,417.964,171.302,33.069,156.192
C06243=1053.801,112.305,417.984,171.300,33.067,156.191
C06244=1053.795,112.056,418.004,171.299,33.064,156.191
C06245=1053.788,111.807,418.024,171.297,33.062,156.191
C06246=1053.783,111.557,418.043,171.295,33.060,156.190
C06247=1053.777,111.308,418.063,171.294,33.058,156.190
C06248=1053.771,111.060,418.083,171.292,33.055,156.190
C06249=1053.765,110.810,418.102,171.290,33.053,156.189
C06250=1053.758,110.561,418.123,171.289,33.051,156.189
C06251=1053.752,110.276,418.145,171.287,33.048,156.188
C06252=1053.744,109.990,418.167,171.285,33.045,156.188
C06253=1053.738,109.705,418.190,171.283,33.043,156.187
C06254=1053.730,109.420,418.213,171.281,33.040,156.187
C06255=1053.725,109.170,418.232,171.279,33.038,156.187
C06256=1053.719,108.921,418.252,171.277,33.035,156.186
C06257=1053.713,108.673,418.272,171.276,33.034,156.186
C06258=1053.706,108.423,418.291,171.274,33.031,156.186
C06259=1053.700,108.174,418.311,171.272,33.029,156.185
C06260=1053.694,107.924,418.330,171.271,33.027,156.185
C06261=1053.688,107.676,418.350,171.270,33.024,156.184
C06262=1053.682,107.426,418.369,171.268,33.022,156.184
C06263=1053.676,107.177,418.389,171.266,33.020,156.184
C06264=1053.669,106.928,418.408,171.265,33.018,156.183
C06265=1053.663,106.679,418.428,171.263,33.015,156.183
C06266=1053.658,106.429,418.447,171.261,33.013,156.183
C06267=1053.652,106.181,418.467,171.260,33.011,156.182
C06268=1053.646,105.931,418.487,171.258,33.009,156.182
C06269=1053.640,105.682,418.506,171.256,33.006,156.181
C06270=1053.633,105.433,418.525,171.255,33.004,156.181
C06271=1053.627,105.184,418.545,171.253,33.002,156.181
C06272=1053.621,104.934,418.565,171.251,33.000,156.180
C06273=1053.615,104.685,418.585,171.250,32.997,156.180
C06274=1053.610,104.436,418.604,171.248,32.995,156.180
C06275=1053.603,104.188,418.623,171.246,32.993,156.179
C06276=1053.597,103.938,418.642,171.245,32.991,156.179
C06277=1053.591,103.689,418.662,171.243,32.988,156.178
C06278=1053.585,103.440,418.682,171.241,32.986,156.178
C06279=1053.580,103.190,418.701,171.240,32.984,156.178
C06280=1053.573,102.942,418.720,171.238,32.982,156.177
C06281=1053.567,102.692,418.740,171.236,32.979,156.177
C06282=1053.562,102.443,418.759,171.235,32.977,156.177
C06283=1053.556,102.194,418.779,171.233,32.974,156.176
C06284=1053.550,101.945,418.798,171.231,32.972,156.176
C06285=1053.544,101.696,418.817,171.230,32.970,156.175
C06286=1053.538,101.447,418.837,171.228,32.968,156.175
C06287=1053.531,101.197,418.856,171.226,32.965,156.175
C06288=1053.526,100.947,418.875,171.225,32.963,156.174
C06289=1053.520,100.698,418.895,171.223,32.961,156.174
C06290=1053.513,100.449,418.914,171.221,32.959,156.174
C06291=1053.507,100.200,418.933,171.220,32.956,156.173
C06292=1053.501,99.951,418.953,171.218,32.954,156.173
C06293=1053.495,99.702,418.972,171.216,32.952,156.172
C06294=1053.489,99.453,418.991,171.214,32.950,156.172
C06295=1053.483,99.203,419.010,171.213,32.948,156.172
C06296=1053.476,98.955,419.029,171.211,32.945,156.171
C06297=1053.470,98.705,419.048,171.209,32.943,156.171
C06298=1053.465,98.456,419.068,171.208,32.941,156.171
C06299=1053.458,98.207,419.086,171.206,32.939,156.170
C06300=1053.453,97.957,419.106,171.204,32.937,156.170
C06301=1053.446,97.709,419.125,171.203,32.934,156.170
C06302=1053.440,97.460,419.144,171.201,32.932,156.169
C06303=1053.434,97.210,419.163,171.199,32.929,156.169
C06304=1053.428,96.961,419.182,171.198,32.928,156.169
C06305=1053.422,96.712,419.201,171.196,32.925,156.168
C06306=1053.416,96.462,419.220,171.194,32.923,156.168
C06307=1053.409,96.214,419.239,171.193,32.921,156.167
C06308=1053.404,95.965,419.259,171.191,32.918,156.167
C06309=1053.397,95.715,419.277,171.189,32.916,156.167
C06310=1053.391,95.466,419.296,171.188,32.914,156.166
C06311=1053.386,95.217,419.316,171.186,32.912,156.166
C06312=1053.379,94.967,419.334,171.184,32.909,156.166
C06313=1053.374,94.718,419.354,171.183,32.907,156.165
C06314=1053.367,94.469,419.372,171.181,32.905,156.165
C06315=1053.360,94.183,419.395,171.179,32.903,156.165
C06316=1053.353,93.898,419.417,171.177,32.900,156.164
C06317=1053.346,93.613,419.438,171.175,32.897,156.164
C06318=1053.340,93.328,419.460,171.174,32.895,156.163
C06319=1053.333,93.078,419.478,171.172,32.892,156.163
C06320=1053.327,92.829,419.498,171.170,32.890,156.162
C06321=1053.321,92.580,419.516,171.169,32.888,156.162
C06322=1053.315,92.330,419.536,171.167,32.886,156.162
C06323=1053.309,92.081,419.554,171.165,32.883,156.161
C06324=1053.303,91.832,419.573,171.164,32.881,156.161
C06325=1053.297,91.583,419.592,171.162,32.879,156.161
C06326=1053.291,91.333,419.611,171.160,32.877,156.160
C06327=1053.285,91.084,419.630,171.159,32.875,156.160
C06328=1053.280,90.835,419.649,171.158,32.872,156.160
C06329=1053.273,90.586,419.668,171.156,32.870,156.159
C06330=1053.268,90.337,419.687,171.155,32.868,156.159
C06331=1053.261,90.088,419.705,171.153,32.866,156.158
C06332=1053.255,89.839,419.724,171.151,32.863,156.158
C06333=1053.248,89.590,419.743,171.150,32.861,156.158
C06334=1053.243,89.339,419.761,171.148,32.859,156.157
C06335=1053.236,89.090,419.780,171.146,32.856,156.157
C06336=1053.230,88.841,419.799,171.145,32.854,156.157
C06337=1053.224,88.592,419.817,171.143,32.852,156.156
C06338=1053.218,88.343,419.836,171.141,32.850,156.156
C06339=1053.211,88.094,419.855,171.140,32.848,156.156
C06340=1053.205,87.844,419.874,171.138,32.846,156.155
C06341=1053.199,87.595,419.892,171.137,32.843,156.155
C06342=1053.194,87.346,419.911,171.135,32.841,156.155
C06343=1053.187,87.097,419.929,171.133,32.839,156.154
C06344=1053.181,86.848,419.948,171.132,32.837,156.154
C06345=1053.175,86.599,419.966,171.130,32.835,156.153
C06346=1053.169,86.349,419.986,171.128,32.833,156.153
C06347=1053.163,86.099,420.004,171.127,32.830,156.153
C06348=1053.156,85.850,420.022,171.125,32.828,156.152
C06349=1053.150,85.601,420.041,171.123,32.826,156.152
C06350=1053.144,85.353,420.059,171.122,32.824,156.152
C06351=1053.138,85.103,420.078,171.120,32.822,156.151
C06352=1053.132,84.854,420.096,171.118,32.819,156.151
C06353=1053.126,84.604,420.115,171.117,32.817,156.151
C06354=1053.119,84.355,420.134,171.115,32.815,156.150
C06355=1053.114,84.106,420.153,171.113,32.812,156.150
C06356=1053.108,83.856,420.171,171.112,32.811,156.150
C06357=1053.102,83.608,420.189,171.110,32.808,156.149
C06358=1053.095,83.359,420.208,171.108,32.806,156.149
C06359=1053.089,83.109,420.226,171.107,32.804,156.148
C06360=1053.084,82.859,420.245,171.105,32.801,156.148
C06361=1053.077,82.610,420.264,171.104,32.799,156.148
C06362=1053.072,82.361,420.281,171.102,32.797,156.147
C06363=1053.065,82.112,420.300,171.100,32.795,156.147
C06364=1053.059,81.863,420.319,171.099,32.793,156.147
C06365=1053.053,81.613,420.337,171.097,32.790,156.146
C06366=1053.047,81.364,420.356,171.095,32.788,156.146
C06367=1053.041,81.115,420.374,171.094,32.786,156.146
C06368=1053.035,80.866,420.392,171.092,32.784,156.145
C06369=1053.029,80.617,420.411,171.091,32.782,156.145
C06370=1053.022,80.367,420.429,171.090,32.779,156.144
C06371=1053.017,80.118,420.447,171.088,32.777,156.144
C06372=1053.011,79.869,420.466,171.087,32.775,156.144
C06373=1053.005,79.619,420.484,171.085,32.773,156.143
C06374=1052.998,79.370,420.503,171.083,32.770,156.143
C06375=1052.993,79.122,420.521,171.082,32.768,156.143
C06376=1052.986,78.872,420.539,171.080,32.766,156.142
C06377=1052.981,78.623,420.558,171.078,32.763,156.142
C06378=1052.975,78.373,420.576,171.077,32.761,156.142
C06379=1052.967,78.088,420.597,171.075,32.759,156.141
C06380=1052.960,77.802,420.617,171.073,32.756,156.141
C06381=1052.954,77.517,420.639,171.071,32.754,156.140
C06382=1052.946,77.231,420.659,171.069,32.751,156.140
C06383=1052.940,76.982,420.678,171.068,32.749,156.140
C06384=1052.934,76.733,420.695,171.066,32.747,156.139
C06385=1052.928,76.484,420.714,171.064,32.745,156.139
C06386=1052.922,76.234,420.732,171.063,32.742,156.139
C06387=1052.916,75.985,420.750,171.061,32.740,156.138
C06388=1052.910,75.736,420.768,171.059,32.738,156.138
C06389=1052.904,75.486,420.786,171.058,32.736,156.138
C06390=1052.897,75.237,420.805,171.056,32.734,156.137
C06391=1052.891,74.987,420.823,171.054,32.732,156.137
C06392=1052.885,74.739,420.841,171.053,32.729,156.136
C06393=1052.879,74.490,420.858,171.051,32.727,156.136
C06394=1052.872,74.240,420.876,171.049,32.725,156.136
C06395=1052.867,73.991,420.895,171.048,32.723,156.135
C06396=1052.860,73.742,420.913,171.046,32.721,156.135
C06397=1052.854,73.493,420.931,171.045,32.719,156.135
C06398=1052.848,73.243,420.949,171.043,32.716,156.134
C06399=1052.842,72.994,420.967,171.041,32.714,156.134
C06400=1052.836,72.745,420.985,171.040,32.712,156.134
C06401=1052.830,72.495,421.003,171.039,32.709,156.133
C06402=1052.824,72.246,421.021,171.037,32.707,156.133
C06403=1052.818,71.997,421.039,171.036,32.705,156.133
C06404=1052.811,71.747,421.057,171.034,32.703,156.132
C06405=1052.806,71.498,421.074,171.032,32.701,156.132
C06406=1052.799,71.249,421.093,171.031,32.699,156.132
C06407=1052.793,70.999,421.111,171.029,32.696,156.131
C06408=1052.787,70.750,421.129,171.028,32.694,156.131
C06409=1052.781,70.501,421.147,171.026,32.692,156.131
C06410=1052.775,70.252,421.165,171.024,32.690,156.130
C06411=1052.769,70.003,421.183,171.023,32.688,156.130
C06412=1052.763,69.753,421.200,171.021,32.686,156.130
C06413=1052.756,69.504,421.219,171.019,32.683,156.129
C06414=1052.751,69.255,421.236,171.018,32.681,156.129
C06415=1052.744,69.005,421.254,171.016,32.679,156.128
C06416=1052.738,68.756,421.272,171.014,32.676,156.128
C06417=1052.732,68.507,421.289,171.013,32.675,156.128
C06418=1052.726,68.258,421.308,171.011,32.673,156.127
C06419=1052.720,68.009,421.325,171.010,32.671,156.127
C06420=1052.713,67.759,421.343,171.008,32.668,156.127
C06421=1052.707,67.509,421.361,171.006,32.666,156.126
C06422=1052.702,67.260,421.378,171.005,32.664,156.126
C06423=1052.696,67.011,421.396,171.003,32.661,156.126
C06424=1052.688,66.762,421.414,171.001,32.659,156.125
C06425=1052.683,66.513,421.432,171.000,32.657,156.125
C06426=1052.677,66.263,421.450,170.998,32.655,156.125
C06427=1052.670,66.014,421.467,170.996,32.653,156.124
C06428=1052.664,65.765,421.485,170.995,32.651,156.124
C06429=1052.658,65.515,421.502,170.994,32.649,156.124
C06430=1052.653,65.266,421.520,170.992,32.646,156.123
C06431=1052.646,65.016,421.537,170.991,32.644,156.123
C06432=1052.640,64.768,421.556,170.989,32.642,156.123
C06433=1052.634,64.518,421.574,170.988,32.640,156.122
C06434=1052.627,64.269,421.591,170.986,32.638,156.122
C06435=1052.622,64.020,421.608,170.984,32.636,156.122
C06436=1052.615,63.770,421.626,170.983,32.634,156.121
C06437=1052.609,63.521,421.643,170.981,32.632,156.121
C06438=1052.602,63.272,421.661,170.979,32.630,156.121
C06439=1052.596,63.022,421.679,170.978,32.627,156.120
C06440=1052.590,62.773,421.696,170.976,32.625,156.120
C06441=1052.584,62.524,421.714,170.974,32.623,156.120
C06442=1052.577,62.274,421.731,170.973,32.621,156.119
C06443=1052.571,61.989,421.750,170.971,32.618,156.119
C06444=1052.563,61.703,421.770,170.969,32.616,156.119
C06445=1052.556,61.418,421.791,170.967,32.614,156.118
C06446=1052.549,61.132,421.810,170.965,32.611,156.118
C06447=1052.542,60.883,421.828,170.963,32.609,156.117
C06448=1052.536,60.634,421.845,170.962,32.607,156.117
C06449=1052.529,60.384,421.863,170.960,32.605,156.117
C06450=1052.524,60.135,421.880,170.958,32.603,156.117
C06451=1052.517,59.885,421.897,170.957,32.601,156.116
C06452=1052.510,59.636,421.914,170.955,32.598,156.116
C06453=1052.505,59.387,421.932,170.953,32.596,156.115
C06454=1052.498,59.137,421.949,170.953,32.594,156.115
C06455=1052.493,58.888,421.967,170.951,32.592,156.115
C06456=1052.486,58.639,421.984,170.950,32.590,156.115
C06457=1052.479,58.390,422.001,170.948,32.588,156.114
C06458=1052.474,58.140,422.018,170.946,32.586,156.114
C06459=1052.467,57.891,422.035,170.945,32.584,156.113
C06460=1052.461,57.641,422.053,170.943,32.582,156.113
C06461=1052.455,57.392,422.070,170.941,32.580,156.113
C06462=1052.448,57.143,422.087,170.940,32.578,156.113
C06463=1052.443,56.894,422.105,170.938,32.575,156.112
C06464=1052.436,56.644,422.122,170.936,32.573,156.112
C06465=1052.431,56.395,422.139,170.935,32.571,156.112
C06466=1052.424,56.145,422.157,170.933,32.569,156.111
C06467=1052.417,55.897,422.174,170.931,32.567,156.111
C06468=1052.411,55.647,422.191,170.930,32.565,156.110
C06469=1052.405,55.398,422.208,170.928,32.563,156.110
C06470=1052.399,55.148,422.226,170.926,32.561,156.110
C06471=1052.393,54.899,422.243,170.925,32.559,156.110
C06472=1052.386,54.650,422.260,170.923,32.556,156.109
C06473=1052.381,54.400,422.277,170.921,32.554,156.109
C06474=1052.374,54.151,422.294,170.920,32.552,156.109
C06475=1052.368,53.902,422.311,170.918,32.550,156.108
C06476=1052.362,53.652,422.329,170.917,32.548,156.108
C06477=1052.356,53.403,422.345,170.916,32.545,156.107
C06478=1052.350,53.153,422.363,170.914,32.543,156.107
C06479=1052.343,52.904,422.380,170.913,32.541,156.107
C06480=1052.337,52.655,422.396,170.911,32.539,156.107
C06481=1052.331,52.405,422.414,170.909,32.537,156.106
C06482=1052.325,52.157,422.431,170.908,32.535,156.106
C06483=1052.318,51.906,422.448,170.906,32.533,156.106
C06484=1052.313,51.657,422.466,170.904,32.531,156.105
C06485=1052.307,51.409,422.483,170.903,32.529,156.105
C06486=1052.300,51.159,422.499,170.901,32.526,156.104
C06487=1052.295,50.910,422.517,170.899,32.524,156.104
C06488=1052.288,50.660,422.533,170.898,32.522,156.104
C06489=1052.282,50.411,422.550,170.896,32.520,156.104
C06490=1052.276,50.162,422.568,170.894,32.517,156.103
C06491=1052.270,49.912,422.585,170.893,32.515,156.103
C06492=1052.263,49.663,422.601,170.891,32.513,156.103
C06493=1052.258,49.414,422.619,170.889,32.511,156.102
C06494=1052.251,49.164,422.636,170.888,32.509,156.102
C06495=1052.245,48.915,422.653,170.886,32.507,156.101
C06496=1052.239,48.665,422.670,170.885,32.505,156.101
C06497=1052.233,48.416,422.687,170.883,32.503,156.101
C06498=1052.227,48.167,422.703,170.882,32.500,156.100
C06499=1052.221,47.917,422.721,170.881,32.498,156.100
C06500=1052.215,47.668,422.737,170.879,32.496,156.100
C06501=1052.209,47.419,422.754,170.877,32.494,156.100
C06502=1052.203,47.169,422.771,170.876,32.492,156.099
C06503=1052.197,46.920,422.788,170.874,32.489,156.099
C06504=1052.191,46.671,422.805,170.872,32.487,156.098
C06505=1052.185,46.421,422.822,170.871,32.485,156.098
C06506=1052.179,46.171,422.839,170.869,32.483,156.098
C06507=1052.172,45.885,422.859,170.867,32.481,156.097
C06508=1052.165,45.601,422.878,170.865,32.478,156.097
C06509=1052.158,45.314,422.897,170.863,32.475,156.097
C06510=1052.151,45.028,422.917,170.862,32.474,156.096
C06511=1052.145,44.779,422.933,170.860,32.471,156.096
C06512=1052.139,44.530,422.950,170.858,32.469,156.096
C06513=1052.132,44.280,422.967,170.857,32.467,156.095
C06514=1052.127,44.030,422.984,170.855,32.464,156.095
C06515=1052.121,43.782,423.001,170.853,32.462,156.095
C06516=1052.115,43.532,423.017,170.852,32.460,156.094
C06517=1052.108,43.283,423.034,170.851,32.458,156.094
C06518=1052.102,43.033,423.051,170.849,32.456,156.094
C06519=1052.097,42.784,423.067,170.848,32.454,156.093
C06520=1052.090,42.534,423.085,170.846,32.452,156.093
C06521=1052.084,42.285,423.101,170.844,32.449,156.093
C06522=1052.078,42.036,423.117,170.843,32.448,156.092
C06523=1052.072,41.787,423.134,170.841,32.445,156.092
C06524=1052.065,41.537,423.151,170.839,32.443,156.092
C06525=1052.059,41.288,423.167,170.838,32.442,156.091
C06526=1052.053,41.039,423.184,170.836,32.439,156.091
C06527=1052.047,40.789,423.201,170.834,32.437,156.091
C06528=1052.041,40.539,423.217,170.833,32.435,156.090
C06529=1052.035,40.290,423.233,170.831,32.433,156.090
C06530=1052.028,40.041,423.250,170.829,32.431,156.090
C06531=1052.022,39.791,423.267,170.828,32.429,156.089
C06532=1052.016,39.542,423.283,170.826,32.427,156.089
C06533=1052.010,39.293,423.300,170.824,32.424,156.089
C06534=1052.004,39.044,423.316,170.823,32.422,156.088
C06535=1051.997,38.794,423.333,170.821,32.420,156.088
C06536=1051.991,38.544,423.349,170.820,32.418,156.088
C06537=1051.985,38.295,423.365,170.819,32.416,156.087
C06538=1051.980,38.046,423.383,170.817,32.414,156.087
C06539=1051.974,37.797,423.399,170.815,32.411,156.087
C06540=1051.966,37.547,423.415,170.814,32.409,156.086
C06541=1051.960,37.298,423.432,170.812,32.407,156.086
C06542=1051.955,37.048,423.448,170.810,32.405,156.086
C06543=1051.949,36.799,423.464,170.809,32.403,156.086
C06544=1051.942,36.550,423.481,170.807,32.401,156.085
C06545=1051.936,36.300,423.498,170.805,32.399,156.085
C06546=1051.930,36.051,423.514,170.804,32.397,156.085
C06547=1051.923,35.802,423.530,170.802,32.395,156.084
C06548=1051.917,35.552,423.546,170.800,32.393,156.084
C06549=1051.911,35.302,423.562,170.798,32.391,156.084
C06550=1051.905,35.053,423.579,170.797,32.389,156.083
C06551=1051.899,34.804,423.595,170.795,32.387,156.083
C06552=1051.893,34.554,423.611,170.793,32.385,156.083
C06553=1051.885,34.305,423.628,170.792,32.383,156.082
C06554=1051.879,34.056,423.644,170.791,32.381,156.082
C06555=1051.873,33.807,423.660,170.789,32.379,156.082
C06556=1051.867,33.557,423.677,170.788,32.376,156.081
C06557=1051.861,33.308,423.693,170.786,32.374,156.081
C06558=1051.854,33.058,423.709,170.784,32.372,156.081
C06559=1051.848,32.809,423.725,170.783,32.370,156.081
C06560=1051.842,32.559,423.742,170.781,32.368,156.080
C06561=1051.836,32.310,423.758,170.779,32.366,156.080
C06562=1051.830,32.061,423.774,170.778,32.364,156.080
C06563=1051.824,31.811,423.790,170.776,32.362,156.079
C06564=1051.817,31.562,423.806,170.774,32.360,156.079
C06565=1051.811,31.312,423.823,170.773,32.358,156.079
C06566=1051.805,31.063,423.839,170.771,32.356,156.078
C06567=1051.799,30.814,423.855,170.769,32.354,156.078
C06568=1051.793,30.564,423.871,170.767,32.352,156.078
C06569=1051.787,30.315,423.887,170.766,32.350,156.078
C06570=1051.781,30.066,423.903,170.764,32.348,156.077
C06571=1051.773,29.780,423.922,170.763,32.345,156.077
C06572=1051.766,29.494,423.940,170.761,32.343,156.077
C06573=1051.759,29.207,423.958,170.759,32.341,156.076
C06574=1051.753,28.922,423.976,170.757,32.338,156.076
C06575=1051.747,28.672,423.993,170.756,32.336,156.075
C06576=1051.740,28.422,424.009,170.754,32.334,156.075
C06577=1051.733,28.173,424.025,170.752,32.332,156.075
C06578=1051.727,27.924,424.041,170.751,32.330,156.074
C06579=1051.721,27.675,424.057,170.749,32.328,156.074
C06580=1051.715,27.425,424.073,170.747,32.326,156.074
C06581=1051.709,27.176,424.089,170.745,32.324,156.074
C06582=1051.703,26.926,424.105,170.744,32.322,156.073
C06583=1051.696,26.677,424.121,170.742,32.320,156.073
C06584=1051.690,26.428,424.137,170.740,32.318,156.073
C06585=1051.683,26.178,424.153,170.739,32.316,156.072
C06586=1051.678,25.928,424.168,170.737,32.314,156.072
C06587=1051.672,25.679,424.185,170.736,32.312,156.072
C06588=1051.665,25.430,424.200,170.734,32.310,156.072
C06589=1051.659,25.180,424.217,170.733,32.308,156.071
C06590=1051.652,24.931,424.232,170.731,32.306,156.071
C06591=1051.647,24.681,424.248,170.729,32.304,156.071
C06592=1051.640,24.432,424.263,170.728,32.302,156.070
C06593=1051.634,24.183,424.280,170.726,32.300,156.070
C06594=1051.628,23.934,424.296,170.724,32.298,156.070
C06595=1051.622,23.684,424.311,170.723,32.296,156.069
C06596=1051.616,23.435,424.327,170.721,32.294,156.069
C06597=1051.609,23.186,424.343,170.719,32.292,156.069
C06598=1051.603,22.936,424.358,170.717,32.290,156.069
C06599=1051.597,22.687,424.374,170.716,32.288,156.068
C06600=1051.591,22.437,424.390,170.714,32.286,156.068
C06601=1051.585,22.187,424.406,170.712,32.284,156.068
C06602=1051.578,21.938,424.421,170.711,32.282,156.067
C06603=1051.572,21.688,424.438,170.710,32.280,156.067
C06604=1051.565,21.438,424.453,170.708,32.278,156.067
C06605=1051.560,21.189,424.469,170.706,32.276,156.066
C06606=1051.553,20.940,424.485,170.705,32.274,156.066
C06607=1051.547,20.690,424.500,170.703,32.272,156.066
C06608=1051.540,20.441,424.516,170.701,32.270,156.066
C06609=1051.535,20.192,424.532,170.700,32.268,156.065
C06610=1051.528,19.942,424.547,170.698,32.266,156.065
C06611=1051.522,19.693,424.564,170.696,32.264,156.065
C06612=1051.516,19.443,424.579,170.694,32.261,156.064
C06613=1051.510,19.194,424.595,170.693,32.260,156.064
C06614=1051.503,18.944,424.610,170.691,32.258,156.064
C06615=1051.497,18.695,424.625,170.689,32.256,156.064
C06616=1051.491,18.446,424.642,170.687,32.254,156.063
C06617=1051.484,18.196,424.657,170.686,32.252,156.063
C06618=1051.479,17.947,424.672,170.684,32.250,156.063
C06619=1051.473,17.698,424.687,170.683,32.248,156.062
C06620=1051.466,17.449,424.703,170.681,32.246,156.062
C06621=1051.460,17.199,424.719,170.680,32.244,156.062
C06622=1051.454,16.950,424.734,170.678,32.242,156.061
C06623=1051.448,16.700,424.750,170.676,32.240,156.061
C06624=1051.441,16.451,424.766,170.675,32.238,156.061
C06625=1051.435,16.201,424.780,170.673,32.236,156.061
C06626=1051.429,15.952,424.797,170.671,32.234,156.060
C06627=1051.423,15.702,424.812,170.669,32.232,156.060
C06628=1051.417,15.452,424.827,170.668,32.230,156.060
C06629=1051.410,15.203,424.843,170.666,32.228,156.059
C06630=1051.404,14.953,424.858,170.664,32.226,156.059
C06631=1051.398,14.704,424.874,170.662,32.224,156.059
C06632=1051.392,14.454,424.889,170.661,32.222,156.059
C06633=1051.386,14.205,424.905,170.659,32.220,156.058
C06634=1051.379,13.955,424.920,170.658,32.218,156.058
C06635=1051.372,13.671,424.938,170.656,32.216,156.058
C06636=1051.365,13.387,424.954,170.654,32.214,156.057
C06637=1051.357,13.101,424.972,170.652,32.212,156.057
C06638=1051.350,12.817,424.989,170.650,32.210,156.057
C06639=1051.343,12.568,425.005,170.648,32.207,156.056
C06640=1051.338,12.318,425.020,170.647,32.206,156.056
C06641=1051.331,12.068,425.035,170.645,32.204,156.056
C06642=1051.325,11.819,425.051,170.643,32.202,156.056
C06643=1051.318,11.570,425.066,170.641,32.200,156.055
C06644=1051.313,11.321,425.081,170.640,32.198,156.055
C06645=1051.306,11.072,425.096,170.638,32.196,156.055
C06646=1051.300,10.822,425.111,170.636,32.194,156.055
C06647=1051.294,10.572,425.127,170.634,32.192,156.054
C06648=1051.288,10.322,425.142,170.634,32.190,156.054
C06649=1051.281,10.073,425.157,170.632,32.189,156.054
C06650=1051.274,9.824,425.172,170.630,32.187,156.054
C06651=1051.268,9.574,425.187,170.628,32.185,156.053
C06652=1051.262,9.324,425.202,170.626,32.183,156.053
C06653=1051.256,9.076,425.217,170.625,32.181,156.053
C06654=1051.250,8.826,425.233,170.623,32.179,156.052
C06655=1051.244,8.576,425.248,170.621,32.177,156.052
C06656=1051.237,8.327,425.263,170.619,32.175,156.052
C06657=1051.231,8.077,425.278,170.618,32.173,156.052
C06658=1051.224,7.828,425.294,170.616,32.172,156.051
C06659=1051.218,7.578,425.308,170.614,32.170,156.051
C06660=1051.212,7.329,425.323,170.612,32.168,156.051
C06661=1051.206,7.080,425.338,170.611,32.166,156.050
C06662=1051.199,6.830,425.353,170.610,32.164,156.050
C06663=1051.194,6.580,425.368,170.608,32.162,156.050
C06664=1051.187,6.331,425.384,170.606,32.160,156.050
C06665=1051.180,6.081,425.399,170.604,32.158,156.049
C06666=1051.175,5.832,425.414,170.603,32.157,156.049
C06667=1051.168,5.583,425.429,170.601,32.154,156.049
C06668=1051.162,5.333,425.444,170.599,32.152,156.049
C06669=1051.156,5.083,425.458,170.597,32.150,156.048
C06670=1051.149,4.834,425.473,170.596,32.148,156.048
C06671=1051.143,4.585,425.488,170.594,32.147,156.048
C06672=1051.137,4.335,425.503,170.592,32.145,156.048
C06673=1051.131,4.086,425.518,170.590,32.143,156.047
C06674=1051.125,3.836,425.534,170.588,32.141,156.047
C06675=1051.119,3.587,425.549,170.587,32.139,156.047
C06676=1051.112,3.338,425.564,170.586,32.137,156.046
C06677=1051.106,3.088,425.579,170.584,32.135,156.046
C06678=1051.100,2.838,425.594,170.582,32.133,156.046
C06679=1051.094,2.589,425.608,170.580,32.132,156.046
C06680=1051.088,2.340,425.623,170.579,32.130,156.045
C06681=1051.081,2.090,425.638,170.577,32.128,156.045
C06682=1051.075,1.840,425.653,170.575,32.125,156.045
C06683=1051.069,1.591,425.668,170.573,32.124,156.045
C06684=1051.063,1.342,425.683,170.572,32.122,156.044
C06685=1051.056,1.092,425.697,170.570,32.120,156.044
C06686=1051.050,0.843,425.712,170.568,32.118,156.044
C06687=1051.044,0.593,425.727,170.566,32.116,156.044
C06688=1051.038,0.344,425.742,170.564,32.114,156.043
C06689=1051.032,0.094,425.757,170.563,32.112,156.043
C06690=1051.026,-0.155,425.772,170.562,32.110,156.043
C06691=1051.020,-0.405,425.787,170.560,32.108,156.042
C06692=1051.014,-0.655,425.801,170.558,32.107,156.042
C06693=1051.008,-0.904,425.816,170.556,32.105,156.042
C06694=1051.002,-1.154,425.831,170.555,32.103,156.042
C06695=1050.995,-1.403,425.846,170.553,32.101,156.041
C06696=1050.989,-1.652,425.860,170.551,32.099,156.041
C06697=1050.983,-1.902,425.875,170.549,32.097,156.041
C06698=1050.977,-2.152,425.890,170.547,32.095,156.041
C06699=1050.970,-2.434,425.907,170.545,32.093,156.040
C06700=1050.963,-2.717,425.923,170.543,32.091,156.040
C06701=1050.956,-2.999,425.940,170.541,32.089,156.040
C06702=1050.949,-3.281,425.957,170.540,32.087,156.039
C06703=1050.943,-3.532,425.971,170.539,32.085,156.039
C06704=1050.937,-3.781,425.986,170.537,32.083,156.039
C06705=1050.930,-4.031,426.001,170.535,32.081,156.039
C06706=1050.924,-4.280,426.015,170.533,32.079,156.038
C06707=1050.918,-4.530,426.029,170.531,32.078,156.038
C06708=1050.911,-4.780,426.044,170.529,32.075,156.038
C06709=1050.906,-5.029,426.059,170.528,32.074,156.038
C06710=1050.899,-5.278,426.073,170.526,32.072,156.037
C06711=1050.892,-5.528,426.087,170.524,32.071,156.037
C06712=1050.887,-5.777,426.102,170.522,32.068,156.037
C06713=1050.880,-6.027,426.116,170.520,32.066,156.037
C06714=1050.873,-6.276,426.131,170.518,32.065,156.036
C06715=1050.868,-6.526,426.145,170.517,32.063,156.036
C06716=1050.861,-6.775,426.160,170.516,32.061,156.036
C06717=1050.854,-7.025,426.174,170.514,32.059,156.036
C06718=1050.849,-7.274,426.188,170.512,32.058,156.035
C06719=1050.842,-7.524,426.203,170.510,32.056,156.035
C06720=1050.837,-7.773,426.218,170.508,32.054,156.035
C06721=1050.830,-8.023,426.231,170.507,32.052,156.035
C06722=1050.823,-8.273,426.246,170.505,32.050,156.034
C06723=1050.818,-8.522,426.261,170.503,32.049,156.034
C06724=1050.811,-8.772,426.274,170.501,32.047,156.034
C06725=1050.805,-9.020,426.289,170.499,32.045,156.034
C06726=1050.799,-9.270,426.304,170.497,32.043,156.033
C06727=1050.793,-9.520,426.318,170.495,32.042,156.033
C06728=1050.786,-9.769,426.332,170.494,32.040,156.033
C06729=1050.780,-10.019,426.346,170.493,32.038,156.033
C06730=1050.774,-10.268,426.361,170.491,32.036,156.032
C06731=1050.767,-10.518,426.375,170.489,32.034,156.032
C06732=1050.762,-10.767,426.389,170.487,32.033,156.032
C06733=1050.755,-11.017,426.404,170.485,32.030,156.032
C06734=1050.748,-11.267,426.418,170.484,32.029,156.032
C06735=1050.743,-11.516,426.432,170.482,32.027,156.031
C06736=1050.736,-11.766,426.446,170.480,32.026,156.031
C06737=1050.730,-12.015,426.460,170.478,32.023,156.031
C06738=1050.724,-12.264,426.475,170.476,32.022,156.031
C06739=1050.718,-12.514,426.489,170.474,32.020,156.030
C06740=1050.711,-12.763,426.504,170.472,32.018,156.030
C06741=1050.705,-13.013,426.517,170.471,32.016,156.030
C06742=1050.699,-13.262,426.532,170.470,32.014,156.030
C06743=1050.693,-13.512,426.546,170.468,32.013,156.029
C06744=1050.687,-13.761,426.561,170.466,32.011,156.029
C06745=1050.681,-14.011,426.575,170.464,32.009,156.029
C06746=1050.674,-14.261,426.588,170.462,32.007,156.029
C06747=1050.668,-14.510,426.603,170.460,32.006,156.028
C06748=1050.662,-14.760,426.617,170.459,32.004,156.028
C06749=1050.656,-15.009,426.631,170.457,32.002,156.028
C06750=1050.650,-15.259,426.645,170.455,32.000,156.028
C06751=1050.643,-15.508,426.659,170.453,31.999,156.027
C06752=1050.637,-15.758,426.673,170.451,31.997,156.027
C06753=1050.631,-16.007,426.687,170.449,31.995,156.027
C06754=1050.625,-16.257,426.702,170.448,31.994,156.027
C06755=1050.618,-16.506,426.715,170.446,31.992,156.027
C06756=1050.612,-16.757,426.729,170.445,31.990,156.026
C06757=1050.606,-17.005,426.743,170.443,31.989,156.026
C06758=1050.600,-17.255,426.757,170.441,31.987,156.026
C06759=1050.593,-17.504,426.771,170.439,31.985,156.026
C06760=1050.586,-17.754,426.785,170.437,31.983,156.025
C06761=1050.581,-18.004,426.799,170.435,31.982,156.025
C06762=1050.574,-18.254,426.812,170.433,31.980,156.025
C06763=1050.567,-18.535,426.828,170.431,31.978,156.025
C06764=1050.560,-18.816,426.844,170.429,31.976,156.025
C06765=1050.553,-19.097,426.860,170.427,31.974,156.024
C06766=1050.546,-19.378,426.875,170.425,31.972,156.024
C06767=1050.539,-19.627,426.890,170.424,31.971,156.024
C06768=1050.533,-19.877,426.903,170.422,31.969,156.024
C06769=1050.528,-20.126,426.917,170.420,31.967,156.023
C06770=1050.521,-20.376,426.931,170.418,31.965,156.023
C06771=1050.515,-20.625,426.945,170.416,31.964,156.023
C06772=1050.508,-20.875,426.959,170.414,31.962,156.023
C06773=1050.503,-21.125,426.973,170.413,31.960,156.022
C06774=1050.496,-21.375,426.986,170.411,31.959,156.022
C06775=1050.489,-21.623,427.000,170.409,31.957,156.022
C06776=1050.484,-21.873,427.014,170.407,31.955,156.022
C06777=1050.477,-22.123,427.028,170.405,31.954,156.022
C06778=1050.471,-22.372,427.041,170.403,31.952,156.021
C06779=1050.465,-22.622,427.055,170.402,31.950,156.021
C06780=1050.459,-22.872,427.068,170.400,31.949,156.021
C06781=1050.453,-23.121,427.083,170.398,31.947,156.021
C06782=1050.446,-23.371,427.097,170.396,31.945,156.021
C06783=1050.440,-23.620,427.110,170.395,31.944,156.020
C06784=1050.434,-23.869,427.124,170.393,31.942,156.020
C06785=1050.427,-24.119,427.137,170.391,31.940,156.020
C06786=1050.422,-24.369,427.151,170.389,31.939,156.020
C06787=1050.416,-24.618,427.165,170.387,31.937,156.019
C06788=1050.409,-24.868,427.179,170.385,31.935,156.019
C06789=1050.403,-25.117,427.193,170.383,31.934,156.019
C06790=1050.397,-25.366,427.206,170.381,31.931,156.019
C06791=1050.390,-25.616,427.220,170.380,31.930,156.019
C06792=1050.385,-25.866,427.234,170.378,31.929,156.018
C06793=1050.378,-26.115,427.247,170.376,31.926,156.018
C06794=1050.372,-26.365,427.260,170.374,31.925,156.018
C06795=1050.366,-26.615,427.274,170.373,31.924,156.018
C06796=1050.360,-26.864,427.288,170.371,31.922,156.018
C06797=1050.353,-27.114,427.301,170.369,31.920,156.017
C06798=1050.347,-27.363,427.315,170.367,31.918,156.017
C06799=1050.341,-27.613,427.328,170.365,31.917,156.017
C06800=1050.335,-27.863,427.342,170.363,31.916,156.017
C06801=1050.328,-28.112,427.355,170.361,31.914,156.017
C06802=1050.322,-28.361,427.369,170.359,31.912,156.016
C06803=1050.315,-28.611,427.382,170.357,31.910,156.016
C06804=1050.309,-28.860,427.395,170.356,31.909,156.016
C06805=1050.303,-29.110,427.409,170.354,31.907,156.016
C06806=1050.297,-29.360,427.423,170.352,31.906,156.016
C06807=1050.291,-29.609,427.436,170.350,31.905,156.015
C06808=1050.284,-29.859,427.450,170.348,31.902,156.015
C06809=1050.278,-30.109,427.463,170.346,31.901,156.015
C06810=1050.272,-30.358,427.476,170.344,31.899,156.015
C06811=1050.265,-30.608,427.489,170.343,31.898,156.015
C06812=1050.259,-30.857,427.502,170.341,31.897,156.014
C06813=1050.252,-31.107,427.516,170.339,31.895,156.014
C06814=1050.246,-31.356,427.529,170.337,31.893,156.014
C06815=1050.241,-31.606,427.543,170.335,31.892,156.014
C06816=1050.234,-31.856,427.557,170.334,31.890,156.014
C06817=1050.228,-32.105,427.570,170.332,31.889,156.013
C06818=1050.222,-32.355,427.582,170.330,31.887,156.013
C06819=1050.216,-32.604,427.596,170.328,31.886,156.013
C06820=1050.209,-32.854,427.609,170.326,31.884,156.013
C06821=1050.203,-33.103,427.623,170.324,31.882,156.013
C06822=1050.196,-33.353,427.636,170.322,31.880,156.013
C06823=1050.190,-33.602,427.648,170.320,31.879,156.012
C06824=1050.184,-33.852,427.662,170.318,31.877,156.012
C06825=1050.177,-34.102,427.675,170.316,31.876,156.012
C06826=1050.172,-34.351,427.689,170.314,31.875,156.012
C06827=1050.165,-34.631,427.704,170.312,31.872,156.012
C06828=1050.158,-34.911,427.719,170.311,31.871,156.011
C06829=1050.151,-35.192,427.733,170.309,31.869,156.011
C06830=1050.144,-35.472,427.748,170.306,31.867,156.011
C06831=1050.137,-35.722,427.761,170.304,31.866,156.011
C06832=1050.131,-35.971,427.775,170.302,31.864,156.011
C06833=1050.125,-36.221,427.787,170.301,31.863,156.010
C06834=1050.120,-36.471,427.801,170.299,31.861,156.010
C06835=1050.113,-36.720,427.814,170.297,31.860,156.010
C06836=1050.107,-36.969,427.827,170.295,31.858,156.010
C06837=1050.101,-37.220,427.840,170.293,31.856,156.010
C06838=1050.094,-37.469,427.854,170.291,31.855,156.009
C06839=1050.088,-37.719,427.867,170.289,31.853,156.009
C06840=1050.082,-37.968,427.880,170.288,31.852,156.009
C06841=1050.076,-38.218,427.893,170.286,31.850,156.009
C06842=1050.070,-38.467,427.906,170.284,31.849,156.009
C06843=1050.064,-38.717,427.919,170.282,31.847,156.009
C06844=1050.057,-38.967,427.932,170.280,31.846,156.008
C06845=1050.051,-39.217,427.945,170.278,31.844,156.008
C06846=1050.044,-39.466,427.957,170.276,31.843,156.008
C06847=1050.038,-39.715,427.971,170.274,31.841,156.008
C06848=1050.032,-39.965,427.983,170.272,31.840,156.008
C06849=1050.026,-40.214,427.997,170.270,31.838,156.008
C06850=1050.019,-40.465,428.009,170.268,31.837,156.007
C06851=1050.013,-40.714,428.023,170.266,31.835,156.007
C06852=1050.007,-40.964,428.035,170.265,31.834,156.007
C06853=1050.000,-41.213,428.048,170.263,31.832,156.007
C06854=1049.994,-41.463,428.061,170.261,31.831,156.007
C06855=1049.988,-41.712,428.074,170.259,31.830,156.007
C06856=1049.982,-41.962,428.086,170.257,31.829,156.006
C06857=1049.975,-42.211,428.099,170.255,31.827,156.006
C06858=1049.969,-42.461,428.112,170.253,31.826,156.006
C06859=1049.963,-42.711,428.125,170.251,31.824,156.006
C06860=1049.957,-42.960,428.138,170.249,31.823,156.006
C06861=1049.951,-43.210,428.151,170.247,31.821,156.006
C06862=1049.945,-43.460,428.164,170.245,31.820,156.005
C06863=1049.938,-43.709,428.176,170.243,31.818,156.005
C06864=1049.932,-43.958,428.189,170.242,31.817,156.005
C06865=1049.926,-44.208,428.202,170.240,31.815,156.005
C06866=1049.920,-44.458,428.215,170.238,31.814,156.005
C06867=1049.913,-44.707,428.227,170.236,31.813,156.005
C06868=1049.907,-44.956,428.240,170.234,31.811,156.004
C06869=1049.901,-45.206,428.252,170.232,31.810,156.004
C06870=1049.895,-45.456,428.266,170.230,31.808,156.004
C06871=1049.889,-45.705,428.278,170.228,31.807,156.004
C06872=1049.882,-45.955,428.290,170.226,31.805,156.004
C06873=1049.876,-46.204,428.303,170.224,31.804,156.004
C06874=1049.870,-46.454,428.316,170.222,31.802,156.003
C06875=1049.864,-46.703,428.329,170.220,31.801,156.003
C06876=1049.857,-46.953,428.341,170.219,31.800,156.003
C06877=1049.851,-47.203,428.354,170.217,31.798,156.003
C06878=1049.845,-47.452,428.367,170.215,31.797,156.003
C06879=1049.839,-47.702,428.380,170.213,31.795,156.003
C06880=1049.833,-47.952,428.392,170.211,31.794,156.003
C06881=1049.826,-48.201,428.405,170.209,31.792,156.002
C06882=1049.820,-48.451,428.417,170.206,31.791,156.002
C06883=1049.814,-48.701,428.430,170.204,31.790,156.002
C06884=1049.808,-48.951,428.443,170.202,31.788,156.002
C06885=1049.802,-49.199,428.455,170.200,31.787,156.002
C06886=1049.796,-49.449,428.468,170.198,31.785,156.002
C06887=1049.790,-49.699,428.480,170.196,31.784,156.002
C06888=1049.784,-49.949,428.493,170.195,31.782,156.001
C06889=1049.777,-50.198,428.506,170.193,31.782,156.001
C06890=1049.771,-50.448,428.518,170.191,31.780,156.001
C06891=1049.764,-50.729,428.532,170.189,31.779,156.001
C06892=1049.756,-51.010,428.546,170.187,31.777,156.001
C06893=1049.749,-51.291,428.560,170.184,31.775,156.001
C06894=1049.742,-51.571,428.574,170.182,31.774,156.000
C06895=1049.736,-51.821,428.586,170.180,31.773,156.000
C06896=1049.729,-52.070,428.598,170.178,31.772,156.000
C06897=1049.723,-52.320,428.611,170.176,31.771,156.000
C06898=1049.717,-52.570,428.623,170.174,31.769,156.000
C06899=1049.711,-52.820,428.635,170.172,31.768,156.000
C06900=1049.704,-53.069,428.647,170.171,31.767,156.000
C06901=1049.697,-53.318,428.660,170.169,31.765,156.000
C06902=1049.691,-53.568,428.672,170.166,31.764,156.000
C06903=1049.685,-53.818,428.684,170.164,31.763,155.999
C06904=1049.679,-54.068,428.697,170.162,31.761,155.999
C06905=1049.672,-54.317,428.709,170.160,31.760,155.999
C06906=1049.665,-54.567,428.721,170.158,31.759,155.999
C06907=1049.660,-54.817,428.733,170.156,31.758,155.999
C06908=1049.653,-55.066,428.745,170.154,31.757,155.999
C06909=1049.647,-55.316,428.758,170.152,31.755,155.999
C06910=1049.640,-55.566,428.770,170.150,31.754,155.999
C06911=1049.634,-55.814,428.781,170.148,31.753,155.998
C06912=1049.628,-56.064,428.794,170.146,31.752,155.998
C06913=1049.622,-56.314,428.806,170.145,31.750,155.998
C06914=1049.616,-56.564,428.818,170.143,31.749,155.998
C06915=1049.609,-56.813,428.830,170.141,31.748,155.998
C06916=1049.603,-57.063,428.842,170.138,31.746,155.998
C06917=1049.597,-57.313,428.855,170.136,31.745,155.998
C06918=1049.590,-57.562,428.867,170.134,31.744,155.998
C06919=1049.583,-57.812,428.879,170.132,31.743,155.997
C06920=1049.577,-58.062,428.891,170.130,31.741,155.997
C06921=1049.571,-58.311,428.903,170.128,31.741,155.997
C06922=1049.565,-58.561,428.916,170.126,31.739,155.997
C06923=1049.559,-58.810,428.927,170.124,31.738,155.997
C06924=1049.552,-59.060,428.939,170.122,31.737,155.997
C06925=1049.546,-59.310,428.952,170.121,31.736,155.997
C06926=1049.540,-59.559,428.964,170.119,31.734,155.997
C06927=1049.534,-59.809,428.975,170.117,31.733,155.997
C06928=1049.528,-60.059,428.987,170.114,31.732,155.996
C06929=1049.521,-60.308,428.999,170.112,31.731,155.996
C06930=1049.515,-60.558,429.011,170.110,31.729,155.996
C06931=1049.509,-60.808,429.024,170.108,31.729,155.996
C06932=1049.502,-61.057,429.036,170.106,31.727,155.996
C06933=1049.496,-61.306,429.047,170.104,31.726,155.996
C06934=1049.490,-61.556,429.060,170.102,31.725,155.996
C06935=1049.484,-61.806,429.071,170.100,31.724,155.996
C06936=1049.477,-62.056,429.083,170.098,31.722,155.996
C06937=1049.472,-62.305,429.095,170.096,31.721,155.995
C06938=1049.465,-62.554,429.107,170.095,31.720,155.995
C06939=1049.459,-62.804,429.119,170.092,31.719,155.995
C06940=1049.453,-63.055,429.131,170.090,31.717,155.995
C06941=1049.446,-63.304,429.143,170.088,31.716,155.995
C06942=1049.440,-63.553,429.155,170.086,31.715,155.995
C06943=1049.434,-63.803,429.167,170.084,31.714,155.995
C06944=1049.428,-64.053,429.178,170.082,31.713,155.995
C06945=1049.421,-64.303,429.190,170.080,31.712,155.995
C06946=1049.416,-64.552,429.203,170.078,31.710,155.994
C06947=1049.409,-64.801,429.215,170.076,31.709,155.994
C06948=1049.403,-65.052,429.226,170.074,31.708,155.994
C06949=1049.397,-65.300,429.237,170.071,31.707,155.994
C06950=1049.391,-65.550,429.250,170.070,31.706,155.994
C06951=1049.385,-65.800,429.262,170.068,31.704,155.994
C06952=1049.378,-66.050,429.273,170.066,31.704,155.994
C06953=1049.373,-66.299,429.285,170.064,31.702,155.994
C06954=1049.366,-66.549,429.297,170.062,31.701,155.994
C06955=1049.359,-66.832,429.310,170.060,31.700,155.994
C06956=1049.352,-67.114,429.324,170.057,31.699,155.993
C06957=1049.346,-67.395,429.337,170.055,31.697,155.993
C06958=1049.339,-67.677,429.350,170.052,31.695,155.993
C06959=1049.333,-67.927,429.362,170.050,31.695,155.993
C06960=1049.327,-68.177,429.373,170.048,31.694,155.993
C06961=1049.320,-68.426,429.385,170.046,31.692,155.993
C06962=1049.314,-68.676,429.397,170.045,31.691,155.993
C06963=1049.309,-68.926,429.409,170.043,31.690,155.993
C06964=1049.302,-69.175,429.421,170.041,31.689,155.993
C06965=1049.296,-69.425,429.432,170.039,31.688,155.993
C06966=1049.290,-69.674,429.443,170.036,31.686,155.992
C06967=1049.284,-69.924,429.456,170.034,31.686,155.992
C06968=1049.277,-70.174,429.467,170.032,31.685,155.992
C06969=1049.271,-70.423,429.479,170.030,31.683,155.992
C06970=1049.265,-70.673,429.490,170.028,31.682,155.992
C06971=1049.260,-70.923,429.502,170.026,31.681,155.992
C06972=1049.253,-71.173,429.513,170.024,31.680,155.992
C06973=1049.247,-71.422,429.525,170.022,31.679,155.992
C06974=1049.241,-71.672,429.536,170.021,31.677,155.992
C06975=1049.235,-71.922,429.549,170.018,31.676,155.992
C06976=1049.229,-72.171,429.560,170.016,31.676,155.992
C06977=1049.223,-72.421,429.572,170.014,31.674,155.991
C06978=1049.217,-72.670,429.583,170.012,31.673,155.991
C06979=1049.211,-72.920,429.595,170.010,31.672,155.991
C06980=1049.205,-73.170,429.606,170.008,31.671,155.991
C06981=1049.199,-73.419,429.618,170.006,31.670,155.991
C06982=1049.192,-73.669,429.629,170.004,31.669,155.991
C06983=1049.187,-73.919,429.641,170.001,31.667,155.991
C06984=1049.181,-74.169,429.653,169.999,31.666,155.991
C06985=1049.175,-74.418,429.663,169.997,31.666,155.991
C06986=1049.168,-74.668,429.675,169.995,31.665,155.991
C06987=1049.162,-74.917,429.686,169.994,31.664,155.991
C06988=1049.155,-75.167,429.697,169.992,31.663,155.991
C06989=1049.149,-75.417,429.709,169.990,31.662,155.991
C06990=1049.143,-75.666,429.720,169.987,31.660,155.990
C06991=1049.136,-75.916,429.732,169.985,31.659,155.990
C06992=1049.131,-76.165,429.743,169.983,31.659,155.990
C06993=1049.124,-76.415,429.754,169.981,31.658,155.990
C06994=1049.118,-76.664,429.765,169.979,31.657,155.990
C06995=1049.112,-76.915,429.777,169.977,31.656,155.990
C06996=1049.106,-77.164,429.788,169.974,31.655,155.990
C06997=1049.100,-77.414,429.799,169.972,31.654,155.990
C06998=1049.094,-77.663,429.810,169.970,31.653,155.990
C06999=1049.087,-77.913,429.822,169.968,31.652,155.990
C07000=1049.081,-78.163,429.833,169.967,31.651,155.990
C07001=1049.075,-78.412,429.845,169.965,31.650,155.990
C07002=1049.069,-78.663,429.856,169.962,31.649,155.990
C07003=1049.063,-78.912,429.867,169.960,31.648,155.990
C07004=1049.057,-79.162,429.878,169.958,31.647,155.990
C07005=1049.051,-79.411,429.889,169.956,31.646,155.989
C07006=1049.045,-79.661,429.900,169.954,31.645,155.989
C07007=1049.038,-79.911,429.912,169.952,31.644,155.989
C07008=1049.031,-80.161,429.922,169.949,31.643,155.989
C07009=1049.026,-80.410,429.933,169.947,31.642,155.989
C07010=1049.019,-80.660,429.944,169.945,31.642,155.989
C07011=1049.013,-80.909,429.956,169.943,31.641,155.989
C07012=1049.006,-81.159,429.967,169.941,31.640,155.989
C07013=1049.000,-81.409,429.977,169.940,31.639,155.989
C07014=1048.994,-81.659,429.989,169.937,31.638,155.989
C07015=1048.988,-81.908,430.000,169.935,31.637,155.989
C07016=1048.981,-82.158,430.010,169.933,31.637,155.989
C07017=1048.976,-82.408,430.021,169.931,31.636,155.989
C07018=1048.969,-82.657,430.033,169.929,31.635,155.989
C07019=1048.962,-82.942,430.045,169.926,31.634,155.989
C07020=1048.954,-83.226,430.057,169.924,31.633,155.989
C07021=1048.947,-83.510,430.070,169.921,31.632,155.989
C07022=1048.941,-83.794,430.082,169.919,31.631,155.989
C07023=1048.934,-84.044,430.093,169.916,31.630,155.989
C07024=1048.928,-84.293,430.104,169.914,31.629,155.989
C07025=1048.921,-84.543,430.115,169.912,31.628,155.989
C07026=1048.915,-84.793,430.126,169.911,31.627,155.989
C07027=1048.910,-85.042,430.137,169.909,31.627,155.989
C07028=1048.903,-85.292,430.148,169.906,31.626,155.989
C07029=1048.897,-85.541,430.158,169.904,31.625,155.989
C07030=1048.891,-85.792,430.170,169.902,31.624,155.988
C07031=1048.885,-86.041,430.181,169.900,31.623,155.988
C07032=1048.878,-86.290,430.191,169.898,31.623,155.988
C07033=1048.872,-86.541,430.202,169.896,31.622,155.988
C07034=1048.866,-86.790,430.213,169.893,31.621,155.988
C07035=1048.859,-87.041,430.223,169.891,31.620,155.988
C07036=1048.854,-87.290,430.234,169.889,31.620,155.988
C07037=1048.848,-87.540,430.245,169.887,31.619,155.988
C07038=1048.841,-87.789,430.255,169.885,31.618,155.988
C07039=1048.835,-88.039,430.266,169.882,31.617,155.988
C07040=1048.829,-88.288,430.277,169.881,31.616,155.988
C07041=1048.822,-88.538,430.288,169.879,31.616,155.988
C07042=1048.817,-88.788,430.299,169.877,31.615,155.988
C07043=1048.810,-89.038,430.310,169.875,31.614,155.988
C07044=1048.804,-89.287,430.320,169.872,31.613,155.988
C07045=1048.798,-89.537,430.331,169.870,31.612,155.988
C07046=1048.791,-89.786,430.342,169.868,31.612,155.988
C07047=1048.786,-90.037,430.352,169.866,31.611,155.988
C07048=1048.780,-90.286,430.363,169.863,31.610,155.988
C07049=1048.773,-90.535,430.373,169.861,31.609,155.988
C07050=1048.767,-90.785,430.384,169.859,31.609,155.988
C07051=1048.761,-91.035,430.395,169.857,31.608,155.988
C07052=1048.755,-91.284,430.405,169.855,31.607,155.988
C07053=1048.749,-91.535,430.416,169.852,31.606,155.988
C07054=1048.743,-91.784,430.427,169.851,31.605,155.988
C07055=1048.737,-92.034,430.437,169.849,31.605,155.988
C07056=1048.730,-92.284,430.448,169.847,31.604,155.988
C07057=1048.724,-92.533,430.459,169.845,31.603,155.988
C07058=1048.718,-92.783,430.469,169.842,31.602,155.988
C07059=1048.713,-93.033,430.480,169.840,31.602,155.988
C07060=1048.705,-93.282,430.490,169.838,31.601,155.988
C07061=1048.700,-93.532,430.501,169.836,31.600,155.988
C07062=1048.694,-93.782,430.511,169.834,31.600,155.988
C07063=1048.688,-94.031,430.522,169.831,31.599,155.988
C07064=1048.682,-94.281,430.532,169.829,31.598,155.988
C07065=1048.675,-94.531,430.543,169.827,31.598,155.988
C07066=1048.670,-94.781,430.553,169.825,31.597,155.988
C07067=1048.663,-95.030,430.564,169.823,31.596,155.988
C07068=1048.657,-95.279,430.574,169.820,31.596,155.988
C07069=1048.651,-95.530,430.585,169.819,31.595,155.988
C07070=1048.645,-95.779,430.595,169.817,31.594,155.988
C07071=1048.639,-96.029,430.606,169.815,31.594,155.988
C07072=1048.633,-96.279,430.616,169.812,31.593,155.988
C07073=1048.627,-96.528,430.627,169.810,31.592,155.988
C07074=1048.621,-96.778,430.638,169.808,31.591,155.988
C07075=1048.615,-97.028,430.647,169.806,31.591,155.988
C07076=1048.609,-97.278,430.658,169.804,31.590,155.988
C07077=1048.603,-97.527,430.668,169.801,31.589,155.988
C07078=1048.597,-97.777,430.679,169.799,31.588,155.988
C07079=1048.590,-98.027,430.689,169.797,31.588,155.988
C07080=1048.584,-98.277,430.699,169.795,31.588,155.988
C07081=1048.578,-98.526,430.710,169.792,31.587,155.988
C07082=1048.572,-98.776,430.719,169.790,31.587,155.988
C07083=1048.564,-99.063,430.731,169.788,31.586,155.988
C07084=1048.557,-99.349,430.743,169.786,31.585,155.988
C07085=1048.550,-99.636,430.755,169.783,31.584,155.988
C07086=1048.544,-99.922,430.766,169.781,31.584,155.988
C07087=1048.537,-100.171,430.777,169.779,31.583,155.988
C07088=1048.532,-100.421,430.787,169.776,31.583,155.988
C07089=1048.525,-100.671,430.797,169.774,31.582,155.988
C07090=1048.518,-100.921,430.807,169.772,31.581,155.988
C07091=1048.513,-101.171,430.818,169.770,31.581,155.988
C07092=1048.507,-101.420,430.827,169.767,31.580,155.988
C07093=1048.500,-101.670,430.838,169.765,31.580,155.988
C07094=1048.495,-101.920,430.848,169.763,31.579,155.988
C07095=1048.488,-102.170,430.858,169.761,31.579,155.988
C07096=1048.481,-102.419,430.868,169.758,31.578,155.988
C07097=1048.476,-102.669,430.879,169.756,31.577,155.988
C07098=1048.469,-102.919,430.889,169.754,31.577,155.988
C07099=1048.463,-103.168,430.898,169.753,31.576,155.988
C07100=1048.457,-103.418,430.908,169.750,31.576,155.988
C07101=1048.451,-103.668,430.919,169.748,31.576,155.988
C07102=1048.445,-103.917,430.929,169.746,31.575,155.988
C07103=1048.439,-104.167,430.938,169.744,31.574,155.988
C07104=1048.433,-104.417,430.949,169.741,31.574,155.988
C07105=1048.426,-104.667,430.959,169.739,31.573,155.988
C07106=1048.420,-104.917,430.969,169.737,31.573,155.988
C07107=1048.414,-105.166,430.978,169.735,31.573,155.988
C07108=1048.408,-105.416,430.989,169.732,31.572,155.988
C07109=1048.402,-105.666,430.999,169.730,31.571,155.988
C07110=1048.396,-105.915,431.008,169.728,31.571,155.988
C07111=1048.389,-106.165,431.019,169.726,31.571,155.988
C07112=1048.384,-106.415,431.029,169.723,31.570,155.988
C07113=1048.378,-106.664,431.038,169.721,31.570,155.988
C07114=1048.372,-106.914,431.048,169.719,31.569,155.988
C07115=1048.365,-107.163,431.058,169.718,31.568,155.988
C07116=1048.360,-107.414,431.068,169.715,31.568,155.989
C07117=1048.353,-107.663,431.078,169.713,31.568,155.989
C07118=1048.347,-107.913,431.087,169.711,31.567,155.989
C07119=1048.341,-108.162,431.098,169.709,31.567,155.989
C07120=1048.335,-108.412,431.107,169.706,31.566,155.989
C07121=1048.328,-108.662,431.117,169.704,31.566,155.989
C07122=1048.322,-108.912,431.126,169.702,31.566,155.989
C07123=1048.316,-109.161,431.137,169.699,31.565,155.989
C07124=1048.310,-109.411,431.147,169.697,31.565,155.989
C07125=1048.304,-109.661,431.156,169.695,31.565,155.989
C07126=1048.298,-109.911,431.166,169.693,31.564,155.989
C07127=1048.292,-110.160,431.176,169.690,31.563,155.989
C07128=1048.286,-110.410,431.185,169.688,31.563,155.989
C07129=1048.279,-110.659,431.195,169.686,31.563,155.989
C07130=1048.273,-110.909,431.205,169.684,31.563,155.989
C07131=1048.267,-111.159,431.215,169.682,31.562,155.989
C07132=1048.261,-111.409,431.224,169.680,31.562,155.989
C07133=1048.255,-111.659,431.234,169.678,31.562,155.989
C07134=1048.249,-111.909,431.244,169.675,31.561,155.989
C07135=1048.243,-112.159,431.253,169.673,31.561,155.990
C07136=1048.237,-112.408,431.263,169.671,31.560,155.989
C07137=1048.231,-112.658,431.273,169.669,31.560,155.990
C07138=1048.224,-112.907,431.283,169.666,31.559,155.990
C07139=1048.218,-113.157,431.292,169.664,31.559,155.990
C07140=1048.212,-113.407,431.302,169.662,31.559,155.990
C07141=1048.206,-113.657,431.312,169.660,31.559,155.990
C07142=1048.199,-113.906,431.321,169.657,31.558,155.990
C07143=1048.193,-114.156,431.331,169.655,31.558,155.990
C07144=1048.187,-114.406,431.340,169.653,31.558,155.990
C07145=1048.181,-114.656,431.350,169.650,31.557,155.990
C07146=1048.175,-114.906,431.359,169.648,31.557,155.990
C07147=1048.169,-115.134,431.368,169.646,31.557,155.990
C07148=1048.164,-115.362,431.376,169.644,31.556,155.990
C07149=1048.158,-115.590,431.385,169.643,31.556,155.990
C07150=1048.153,-115.819,431.395,169.641,31.556,155.990
C07151=1048.147,-116.047,431.403,169.639,31.556,155.990
C07152=1048.142,-116.275,431.412,169.637,31.555,155.990
C07153=1048.136,-116.504,431.420,169.635,31.555,155.991
C07154=1048.130,-116.732,431.429,169.632,31.555,155.991
C07155=1048.124,-116.982,431.438,169.630,31.554,155.991
C07156=1048.118,-117.232,431.448,169.628,31.554,155.991
C07157=1048.112,-117.482,431.457,169.626,31.554,155.991
C07158=1048.106,-117.731,431.467,169.623,31.554,155.991
C07159=1048.100,-117.980,431.476,169.621,31.554,155.991
C07160=1048.094,-118.230,431.486,169.619,31.554,155.991
C07161=1048.087,-118.480,431.495,169.616,31.553,155.991
C07162=1048.081,-118.730,431.503,169.614,31.553,155.991
C07163=1048.073,-119.058,431.516,169.611,31.552,155.991
C07164=1048.065,-119.386,431.528,169.608,31.553,155.992
C07165=1048.057,-119.715,431.540,169.605,31.552,155.992
C07166=1048.049,-120.043,431.552,169.602,31.552,155.992
C07167=1048.043,-120.293,431.562,169.601,31.552,155.992
C07168=1048.037,-120.543,431.572,169.598,31.551,155.992
C07169=1048.031,-120.792,431.581,169.596,31.551,155.992
C07170=1048.025,-121.042,431.590,169.594,31.551,155.992
C07171=1048.019,-121.292,431.599,169.592,31.551,155.992
C07172=1048.013,-121.542,431.609,169.589,31.551,155.992
C07173=1048.006,-121.792,431.618,169.587,31.550,155.992
C07174=1048.000,-122.041,431.627,169.585,31.550,155.992
C07175=1047.994,-122.291,431.637,169.582,31.550,155.993
C07176=1047.988,-122.541,431.645,169.580,31.550,155.993
C07177=1047.982,-122.791,431.655,169.578,31.550,155.993
C07178=1047.976,-123.041,431.665,169.575,31.549,155.993
C07179=1047.970,-123.289,431.673,169.573,31.550,155.993
C07180=1047.964,-123.540,431.682,169.571,31.549,155.993
C07181=1047.958,-123.790,431.692,169.569,31.549,155.993
C07182=1047.951,-124.039,431.701,169.566,31.549,155.993
C07183=1047.946,-124.289,431.710,169.564,31.549,155.993
C07184=1047.939,-124.539,431.719,169.562,31.549,155.993
C07185=1047.933,-124.788,431.728,169.559,31.549,155.993
C07186=1047.927,-125.039,431.737,169.557,31.549,155.994
C07187=1047.921,-125.289,431.747,169.555,31.549,155.994
C07188=1047.915,-125.537,431.755,169.553,31.548,155.994
C07189=1047.909,-125.788,431.764,169.551,31.549,155.994
C07190=1047.903,-126.038,431.774,169.549,31.548,155.994
C07191=1047.896,-126.287,431.783,169.547,31.548,155.994
C07192=1047.890,-126.537,431.791,169.544,31.548,155.994
C07193=1047.884,-126.787,431.801,169.542,31.548,155.994
C07194=1047.878,-127.037,431.809,169.540,31.548,155.994
C07195=1047.872,-127.286,431.818,169.537,31.548,155.995
C07196=1047.866,-127.536,431.828,169.535,31.548,155.995
C07197=1047.859,-127.786,431.836,169.533,31.548,155.995
C07198=1047.855,-128.035,431.846,169.530,31.548,155.995
C07199=1047.850,-128.285,431.856,169.528,31.547,155.995
C07200=1047.846,-128.534,431.866,169.526,31.545,155.995
C07201=1047.844,-128.785,431.878,169.524,31.544,155.994
C07202=1047.842,-129.035,431.890,169.523,31.541,155.994
C07203=1047.842,-129.285,431.902,169.522,31.538,155.994
C07204=1047.843,-129.536,431.916,169.520,31.535,155.993
C07205=1047.844,-129.786,431.929,169.519,31.532,155.993
C07206=1047.847,-130.035,431.943,169.517,31.528,155.992
C07207=1047.850,-130.287,431.959,169.516,31.522,155.991
C07208=1047.855,-130.537,431.975,169.516,31.518,155.990
C07209=1047.860,-130.788,431.991,169.515,31.512,155.990
C07210=1047.867,-131.038,432.008,169.514,31.506,155.989
C07211=1047.507,-131.061,431.775,169.468,31.680,156.021
C07212=1047.500,-130.811,431.757,169.469,31.686,156.022
C07213=1047.495,-130.561,431.741,169.470,31.692,156.023
C07214=1047.490,-130.310,431.726,169.470,31.697,156.024
C07215=1047.487,-130.060,431.711,169.471,31.701,156.024
C07216=1047.484,-129.810,431.695,169.473,31.705,156.025
C07217=1047.482,-129.559,431.682,169.474,31.709,156.025
C07218=1047.482,-129.309,431.669,169.476,31.712,156.026
C07219=1047.482,-129.058,431.656,169.478,31.715,156.026
C07220=1047.483,-128.808,431.644,169.478,31.717,156.027
C07221=1047.486,-128.558,431.633,169.480,31.719,156.027
C07222=1047.489,-128.308,431.622,169.482,31.721,156.027
C07223=1047.494,-128.059,431.612,169.484,31.721,156.027
C07224=1047.499,-127.809,431.602,169.487,31.722,156.027
C07225=1047.505,-127.559,431.593,169.489,31.722,156.027
C07226=1047.511,-127.310,431.585,169.491,31.722,156.027
C07227=1047.517,-127.060,431.575,169.494,31.722,156.027
C07228=1047.523,-126.810,431.566,169.496,31.722,156.026
C07229=1047.529,-126.561,431.558,169.498,31.722,156.026
C07230=1047.536,-126.311,431.548,169.501,31.722,156.026
C07231=1047.541,-126.061,431.539,169.503,31.722,156.026
C07232=1047.548,-125.811,431.530,169.505,31.722,156.026
C07233=1047.554,-125.562,431.522,169.508,31.722,156.026
C07234=1047.560,-125.312,431.512,169.510,31.722,156.026
C07235=1047.567,-125.062,431.503,169.512,31.722,156.026
C07236=1047.573,-124.812,431.494,169.514,31.722,156.026
C07237=1047.578,-124.563,431.485,169.517,31.723,156.026
C07238=1047.584,-124.313,431.476,169.518,31.723,156.025
C07239=1047.591,-124.063,431.467,169.520,31.722,156.025
C07240=1047.597,-123.813,431.458,169.523,31.723,156.025
C07241=1047.603,-123.564,431.449,169.525,31.723,156.025
C07242=1047.609,-123.314,431.440,169.527,31.723,156.025
C07243=1047.615,-123.064,431.430,169.530,31.723,156.025
C07244=1047.621,-122.814,431.421,169.532,31.723,156.025
C07245=1047.628,-122.564,431.412,169.534,31.724,156.025
C07246=1047.633,-122.315,431.403,169.537,31.723,156.025
C07247=1047.639,-122.065,431.394,169.539,31.724,156.025
C07248=1047.645,-121.815,431.384,169.541,31.724,156.025
C07249=1047.652,-121.565,431.375,169.544,31.724,156.024
C07250=1047.657,-121.315,431.366,169.546,31.724,156.024
C07251=1047.664,-121.066,431.357,169.548,31.724,156.024
C07252=1047.670,-120.816,431.348,169.550,31.724,156.024
C07253=1047.676,-120.567,431.338,169.553,31.725,156.024
C07254=1047.682,-120.317,431.328,169.555,31.725,156.024
C07255=1047.688,-120.066,431.320,169.557,31.725,156.024
C07256=1047.694,-119.817,431.310,169.560,31.725,156.024
C07257=1047.700,-119.567,431.301,169.562,31.725,156.024
C07258=1047.706,-119.318,431.291,169.563,31.726,156.024
C07259=1047.713,-119.068,431.282,169.566,31.726,156.024
C07260=1047.719,-118.818,431.273,169.568,31.726,156.024
C07261=1047.725,-118.569,431.263,169.570,31.726,156.023
C07262=1047.731,-118.318,431.254,169.572,31.726,156.023
C07263=1047.737,-118.069,431.245,169.575,31.726,156.023
C07264=1047.743,-117.819,431.235,169.577,31.727,156.023
C07265=1047.749,-117.569,431.226,169.579,31.727,156.023
C07266=1047.755,-117.320,431.216,169.582,31.727,156.023
C07267=1047.761,-117.070,431.207,169.584,31.728,156.023
C07268=1047.768,-116.820,431.197,169.586,31.728,156.023
C07269=1047.774,-116.570,431.188,169.589,31.728,156.023
C07270=1047.780,-116.320,431.178,169.591,31.728,156.023
C07271=1047.787,-116.071,431.169,169.593,31.728,156.023
C07272=1047.793,-115.785,431.159,169.596,31.729,156.023
C07273=1047.800,-115.500,431.148,169.598,31.729,156.022
C07274=1047.807,-115.214,431.136,169.601,31.729,156.022
C07275=1047.814,-114.929,431.126,169.604,31.730,156.022
C07276=1047.820,-114.679,431.116,169.606,31.730,156.022
C07277=1047.827,-114.430,431.107,169.607,31.730,156.022
C07278=1047.833,-114.180,431.097,169.610,31.731,156.022
C07279=1047.839,-113.930,431.087,169.612,31.731,156.022
C07280=1047.845,-113.680,431.078,169.614,31.731,156.022
C07281=1047.851,-113.430,431.068,169.616,31.731,156.022
